// TIA Portal V18 program export: 17 tag tables, 4 data types, 7 data blocks, 10 code blocks (in call order from the OBs), 10 instance data blocks

VAR_GLOBAL   // PLC tag table "Cabinet_1"
   Sz1_Button_LED_ST25_ST26 AT %Q1100.0 : Bool;
   Sz1_Button_LED_ST26_ST27 AT %Q1100.1 : Bool;
   Sz1_Button_LED_ST24_ST23 AT %Q1100.2 : Bool;
   Sz1_Button_LED_ST23_ST22 AT %Q1100.3 : Bool;
   Sz1_Button_LED_Hyd_Up AT %Q1100.4 : Bool;
   Sz1_Button_LED_Hyd_Down AT %Q1100.5 : Bool;
   Sz1_Button_LED_Air_Up AT %Q1100.6 : Bool;
   Sz1_Button_LED_Air_Down AT %Q1100.7 : Bool;
   Sz1_Button_LED_Wibration AT %Q1101.0 : Bool;
   Sz1_Button_LED_SS_Down AT %Q1101.1 : Bool;
   Sz1_Button_LED_SS_Up AT %Q1101.2 : Bool;
   Sz1_Button_LED_SS_Drive_ST25 AT %Q1101.3 : Bool;
   Sz1_Button_LED_SS_Drive_ST24 AT %Q1101.4 : Bool;
   Sz1_Button_LED_SS_Drive_ST17 AT %Q1101.5 : Bool;
   Sz1_Button_LED_SS_Drive_ST14 AT %Q1101.6 : Bool;
   Reserved AT %Q1101.7 : Bool;
   Sz1_St25_SenA AT %I1100.0 : Bool;
   Sz1_St25_SenB AT %I1100.1 : Bool;
   Sz1_St25_SenC AT %I1100.2 : Bool;
   Sz1_St25_SenD AT %I1100.3 : Bool;
   Sz1_St26_SenA AT %I1100.4 : Bool;
   Sz1_St26_SenB AT %I1100.5 : Bool;
   Sz1_St26_SenC AT %I1100.6 : Bool;
   Sz1_St26_SenD AT %I1100.7 : Bool;
   Sz1_St23_SenA AT %I1101.0 : Bool;
   Sz1_St23_SenB AT %I1101.1 : Bool;
   Sz1_St23_SenC AT %I1101.2 : Bool;
   Sz1_St23_SenD AT %I1101.3 : Bool;
   Sz1_St24_SenA AT %I1101.4 : Bool;
   Sz1_St24_SenB AT %I1101.5 : Bool;
   Sz1_St24_SenC AT %I1101.6 : Bool;
   Sz1_St24_SenD AT %I1101.7 : Bool;
   Sz1_Button_ST25_ST26 AT %I1102.0 : Bool;
   Sz1_Button_ST26_ST27 AT %I1102.1 : Bool;
   Sz1_Button_ST24_ST23 AT %I1102.2 : Bool;
   Sz1_Button_ST23_ST22 AT %I1102.3 : Bool;
   Sz1_Button_Hyd_Up AT %I1102.4 : Bool;
   Sz1_Button_Hyd_Down AT %I1102.5 : Bool;
   Sz1_Button_Air_Up AT %I1102.6 : Bool;
   Sz1_Button_Air_Down AT %I1102.7 : Bool;
   Sz1_Button_Wibration AT %I1103.0 : Bool;
   Sz1_Button_SS_Down AT %I1103.1 : Bool;
   Sz1_Button_SS_Up AT %I1103.2 : Bool;
   Sz1_Button_SS_Drive_ST25 AT %I1103.3 : Bool;
   Sz1_Button_SS_Drive_ST24 AT %I1103.4 : Bool;
   Sz1_Button_SS_Drive_ST17 AT %I1103.5 : Bool;
   Sz1_Button_SS_Drive_ST14 AT %I1103.6 : Bool;
   "Reserved(1)" AT %I1103.7 : Bool;
   Sz1_Button_Wib_ST25 AT %I1104.0 : Bool;
   Sz1_Button_Wib_ST24 AT %I1104.1 : Bool;
   Sz1_Button_Wib_ST23 AT %I1104.2 : Bool;
   Sz1_Button_Centering_ST23 AT %I1104.3 : Bool;
   Sz1_Button_Centering_ST22 AT %I1104.4 : Bool;
   "Reserved(2)" AT %I1104.5 : Bool;
   "Reserved(3)" AT %I1104.6 : Bool;
   "Reserved(4)" AT %I1104.7 : Bool;
   Sz1_Button_LED_Centering_ST23 AT %Q1102.0 : Bool;
   Sz1_Button_LED_Centering_ST22 AT %Q1102.1 : Bool;
   "Reserved(5)" AT %Q1102.2 : Bool;
   "Reserved(6)" AT %Q1102.3 : Bool;
   "Reserved(7)" AT %Q1102.4 : Bool;
   "Reserved(8)" AT %Q1102.5 : Bool;
   "Reserved(9)" AT %Q1102.6 : Bool;
   "Reserved(10)" AT %Q1102.7 : Bool;
   Sz1_Safety1_1 AT %I1150.0 : Bool;
   "Reserved(11)" AT %I1150.1 : Bool;
   "Reserved(12)" AT %I1150.2 : Bool;
   "Reserved(13)" AT %I1150.3 : Bool;
   Sz1_Safety1_2 AT %I1150.4 : Bool;
   "Reserved(14)" AT %I1150.5 : Bool;
   "Reserved(15)" AT %I1150.6 : Bool;
   "Reserved(16)" AT %I1150.7 : Bool;
   "Reserved(17)" AT %I1151.0 : Bool;
   "Reserved(18)" AT %I1151.1 : Bool;
   "Reserved(19)" AT %I1151.2 : Bool;
   "Reserved(20)" AT %I1151.3 : Bool;
   "Reserved(21)" AT %I1151.4 : Bool;
   "Reserved(22)" AT %I1151.5 : Bool;
   "Reserved(23)" AT %I1151.6 : Bool;
   "Reserved(24)" AT %I1151.7 : Bool;
END_VAR

VAR_GLOBAL   // PLC tag table "Cabinet_10"
   Sz10_Button_LED_ST11_ST12 AT %Q2000.0 : Bool;
   Sz10_Button_LED_ST12_ST13 AT %Q2000.1 : Bool;
   "Reserved(146)" AT %Q2000.2 : Bool;
   "Reserved(147)" AT %Q2000.3 : Bool;
   "Reserved(148)" AT %Q2000.4 : Bool;
   "Reserved(149)" AT %Q2000.5 : Bool;
   "Reserved(150)" AT %Q2000.6 : Bool;
   "Reserved(151)" AT %Q2000.7 : Bool;
   Sz10_ST11_SenA AT %I2000.0 : Bool;
   Sz10_ST11_SenB AT %I2000.1 : Bool;
   Sz10_ST11_SenC AT %I2000.2 : Bool;
   Sz10_ST11_SenD AT %I2000.3 : Bool;
   Sz10_ST12_SenA AT %I2000.4 : Bool;
   Sz10_ST12_SenB AT %I2000.5 : Bool;
   Sz10_ST12_SenC AT %I2000.6 : Bool;
   Sz10_ST12_SenD AT %I2000.7 : Bool;
   Sz10_Button_ST11_ST12 AT %I2001.0 : Bool;
   Sz10_Button_ST12_ST13 AT %I2001.1 : Bool;
   "Reserved(152)" AT %I2001.2 : Bool;
   "Reserved(153)" AT %I2001.3 : Bool;
   "Reserved(154)" AT %I2001.4 : Bool;
   "Reserved(155)" AT %I2001.5 : Bool;
   "Reserved(156)" AT %I2001.6 : Bool;
   "Reserved(157)" AT %I2001.7 : Bool;
   Sz10_Safety1_1 AT %I2050.0 : Bool;
   "Reserved(158)" AT %I2050.1 : Bool;
   "Reserved(159)" AT %I2050.2 : Bool;
   "Reserved(160)" AT %I2050.3 : Bool;
   Sz10_Safety1_2 AT %I2050.4 : Bool;
   "Reserved(161)" AT %I2050.5 : Bool;
   "Reserved(162)" AT %I2050.6 : Bool;
   "Reserved(163)" AT %I2050.7 : Bool;
   "Reserved(171)" AT %I2051.0 : Bool;
   "Reserved(170)" AT %I2051.1 : Bool;
   "Reserved(169)" AT %I2051.2 : Bool;
   "Reserved(168)" AT %I2051.3 : Bool;
   "Reserved(167)" AT %I2051.4 : Bool;
   "Reserved(166)" AT %I2051.5 : Bool;
   "Reserved(165)" AT %I2051.6 : Bool;
   "Reserved(164)" AT %I2051.7 : Bool;
END_VAR

VAR_GLOBAL   // PLC tag table "Cabinet_11"
   Sz11_ST13_SenA AT %I2100.0 : Bool;
   Sz11_ST13_SenB AT %I2100.1 : Bool;
   Sz11_ST13_SenC AT %I2100.2 : Bool;
   Sz11_ST13_SenD AT %I2100.3 : Bool;
   Sz11_ST14_SenA AT %I2100.4 : Bool;
   Sz11_ST14_SenB AT %I2100.5 : Bool;
   Sz11_ST14_SenC AT %I2100.6 : Bool;
   Sz11_ST14_SenD AT %I2100.7 : Bool;
   Sz11_ST17_SenA AT %I2101.0 : Bool;
   Sz11_ST17_SenB AT %I2101.1 : Bool;
   Sz11_ST17_SenC AT %I2101.2 : Bool;
   Sz11_ST17_SenD AT %I2101.3 : Bool;
   "Reserved(188)" AT %I2101.4 : Bool;
   "Reserved(189)" AT %I2101.5 : Bool;
   "Reserved(190)" AT %I2101.6 : Bool;
   Sz11_Safety1_1 AT %I2150.0 : Bool;
   "Reserved(173)" AT %I2150.1 : Bool;
   "Reserved(174)" AT %I2150.2 : Bool;
   "Reserved(175)" AT %I2150.3 : Bool;
   Sz11_Safety1_2 AT %I2150.4 : Bool;
   "Reserved(176)" AT %I2150.5 : Bool;
   "Reserved(177)" AT %I2150.6 : Bool;
   "Reserved(178)" AT %I2150.7 : Bool;
   "Reserved(179)" AT %I2151.0 : Bool;
   "Reserved(180)" AT %I2151.1 : Bool;
   "Reserved(181)" AT %I2151.2 : Bool;
   "Reserved(182)" AT %I2151.3 : Bool;
   "Reserved(183)" AT %I2151.4 : Bool;
   "Reserved(184)" AT %I2151.5 : Bool;
   "Reserved(185)" AT %I2151.6 : Bool;
   "Reserved(186)" AT %I2151.7 : Bool;
   Sz11_Button_LED_ST13_ST14 AT %Q2100.0 : Bool;
   "Reserved(187)" AT %I2101.7 : Bool;
   Sz11_Button_LED_SS_Down AT %Q2100.1 : Bool;
   Sz11_Button_LED_SS_Up AT %Q2100.2 : Bool;
   Sz11_Button_LED_SS_Drive_ST14 AT %Q2100.3 : Bool;
   Sz11_Button_LED_SS_Drive_ST17 AT %Q2100.4 : Bool;
   Sz11_Button_LED_SS_Drive_ST24 AT %Q2100.5 : Bool;
   Sz11_Button_LED_SS_Drive_ST25 AT %Q2100.6 : Bool;
   "Reserved(172)" AT %Q2100.7 : Bool;
   Sz11_Button_ST13_ST14 AT %I2102.0 : Bool;
   Sz11_Button_SS_Down AT %I2102.1 : Bool;
   Sz11_Button_SS_Up AT %I2102.2 : Bool;
   Sz11_Button_SS_Drive_ST14 AT %I2102.3 : Bool;
   Sz11_Button_SS_Drive_ST17 AT %I2102.4 : Bool;
   Sz11_Button_SS_Drive_ST24 AT %I2102.5 : Bool;
   Sz11_Button_SS_Drive_ST25 AT %I2102.6 : Bool;
END_VAR

VAR_GLOBAL   // PLC tag table "Cabinet_2"
   Sz2_Button_LED_ST27_ST28 AT %Q1200.0 : Bool;
   Sz2_Button_LED_ST28_ST29 AT %Q1200.1 : Bool;
   Sz2_Button_LED_ST22_ST21 AT %Q1200.2 : Bool;
   Sz2_Button_LED_ST21_ST20 AT %Q1200.3 : Bool;
   Sz2_Button_LED_Centering_ST21 AT %Q1200.4 : Bool;
   Sz2_Button_LED_Centering_ST20 AT %Q1200.5 : Bool;
   "Reserved(25)" AT %Q1200.6 : Bool;
   "Reserved(26)" AT %Q1200.7 : Bool;
   Sz2_ST27_SenA AT %I1200.0 : Bool;
   Sz2_ST27_SenB AT %I1200.1 : Bool;
   Sz2_ST27_SenC AT %I1200.2 : Bool;
   Sz2_ST27_SenD AT %I1200.3 : Bool;
   Sz2_ST28_SenA AT %I1200.4 : Bool;
   Sz2_ST28_SenB AT %I1200.5 : Bool;
   Sz2_ST28_SenC AT %I1200.6 : Bool;
   Sz2_ST28_SenD AT %I1200.7 : Bool;
   Sz2_ST21_SenA AT %I1201.0 : Bool;
   Sz2_ST21_SenB AT %I1201.1 : Bool;
   Sz2_ST21_SenC AT %I1201.2 : Bool;
   Sz2_ST21_SenD AT %I1201.3 : Bool;
   Sz2_ST22_SenA AT %I1201.4 : Bool;
   Sz2_ST22_SenB AT %I1201.5 : Bool;
   Sz2_ST22_SenC AT %I1201.6 : Bool;
   Sz2_ST22_SenD AT %I1201.7 : Bool;
   Sz2_Button_ST27_ST28 AT %I1202.0 : Bool;
   Sz2_Button_ST28_ST29 AT %I1202.1 : Bool;
   Sz2_Button_ST22_ST21 AT %I1202.2 : Bool;
   Sz2_Button_ST21_ST20 AT %I1202.3 : Bool;
   Sz2_Button_Centering_ST21 AT %I1202.4 : Bool;
   Sz2_Button_Centering_ST20 AT %I1202.5 : Bool;
   "Reserved(27)" AT %I1202.6 : Bool;
   "Reserved(28)" AT %I1202.7 : Bool;
   Sz2_Safety_1_1 AT %I1250.0 : Bool;
   Sz2_Safety_1_2 AT %I1250.4 : Bool;
   "Reserved(29)" AT %I1250.1 : Bool;
   "Reserved(30)" AT %I1250.2 : Bool;
   "Reserved(31)" AT %I1250.3 : Bool;
   "Reserved(32)" AT %I1250.5 : Bool;
   "Reserved(33)" AT %I1250.6 : Bool;
   "Reserved(34)" AT %I1250.7 : Bool;
   "Reserved(35)" AT %I1251.0 : Bool;
   "Reserved(36)" AT %I1251.1 : Bool;
   "Reserved(37)" AT %I1251.2 : Bool;
   "Reserved(38)" AT %I1251.3 : Bool;
   "Reserved(39)" AT %I1251.4 : Bool;
   "Reserved(40)" AT %I1251.5 : Bool;
   "Reserved(41)" AT %I1251.6 : Bool;
   "Reserved(42)" AT %I1251.7 : Bool;
END_VAR

VAR_GLOBAL   // PLC tag table "Cabinet_3"
   Sz3_Button_LED_ST29_ST30 AT %Q1300.0 : Bool;
   Sz3_Button_LED_ST30_ST31 AT %Q1300.1 : Bool;
   Sz3_Button_LED_ST18_ST37 AT %Q1300.2 : Bool;
   Sz3_Button_LED_ST19_ST18 AT %Q1300.3 : Bool;
   Sz3_Button_LED_ST20_ST19 AT %Q1300.4 : Bool;
   Sz3_Button_LED_Centering_ST19 AT %Q1300.5 : Bool;
   Sz3_Button_LED_Centering_ST18 AT %Q1300.6 : Bool;
   "Reserved(43)" AT %Q1300.7 : Bool;
   Sz3_ST29_SenA AT %I1300.0 : Bool;
   Sz3_ST29_SenB AT %I1300.1 : Bool;
   Sz3_ST29_SenC AT %I1300.2 : Bool;
   Sz3_ST29_SenD AT %I1300.3 : Bool;
   Sz3_ST30_SenA AT %I1300.4 : Bool;
   Sz3_ST30_SenB AT %I1300.5 : Bool;
   Sz3_ST30_SenC AT %I1300.6 : Bool;
   Sz3_ST30_SenD AT %I1300.7 : Bool;
   Sz3_ST31_SenA AT %I1301.0 : Bool;
   Sz3_ST31_SenB AT %I1301.1 : Bool;
   Sz3_ST31_SenC AT %I1301.2 : Bool;
   Sz3_ST31_SenD AT %I1301.3 : Bool;
   Sz3_ST18_SenA AT %I1301.4 : Bool;
   Sz3_ST18_SenB AT %I1301.5 : Bool;
   Sz3_ST18_SenC AT %I1301.6 : Bool;
   Sz3_ST18_SenD AT %I1301.7 : Bool;
   Sz3_ST19_SenA AT %I1302.0 : Bool;
   Sz3_ST19_SenB AT %I1302.1 : Bool;
   Sz3_ST19_SenC AT %I1302.2 : Bool;
   Sz3_ST19_SenD AT %I1302.3 : Bool;
   Sz3_ST20_SenA AT %I1302.4 : Bool;
   Sz3_ST20_SenB AT %I1302.5 : Bool;
   Sz3_ST20_SenC AT %I1302.6 : Bool;
   Sz3_ST20_SenD AT %I1302.7 : Bool;
   Sz3_Button_ST29_ST30 AT %I1303.0 : Bool;
   Sz3_Button_ST30_ST31 AT %I1303.1 : Bool;
   Sz3_Button_ST31_ST32 AT %I1303.2 : Bool;
   Sz3_Button_ST18_ST37 AT %I1303.3 : Bool;
   Sz3_Button_ST19_ST18 AT %I1303.4 : Bool;
   Sz3_Button_ST20_ST19 AT %I1303.5 : Bool;
   Sz3_Button_Centering_ST19 AT %I1303.6 : Bool;
   Sz3_Button_Centering_ST18 AT %I1303.7 : Bool;
   Sz3_Safety1_1 AT %I1304.0 : Bool;
   "Reserved(44)" AT %I1304.1 : Bool;
   "Reserved(45)" AT %I1304.2 : Bool;
   "Reserved(46)" AT %I1304.3 : Bool;
   Sz3_Safety1_2 AT %I1304.4 : Bool;
   "Reserved(47)" AT %I1304.5 : Bool;
   "Reserved(48)" AT %I1304.6 : Bool;
   "Reserved(49)" AT %I1304.7 : Bool;
   "Reserved(50)" AT %I1305.0 : Bool;
   "Reserved(51)" AT %I1305.1 : Bool;
   "Reserved(52)" AT %I1305.2 : Bool;
   "Reserved(53)" AT %I1305.3 : Bool;
   "Reserved(54)" AT %I1305.4 : Bool;
   "Reserved(55)" AT %I1305.5 : Bool;
   "Reserved(56)" AT %I1305.6 : Bool;
   "Reserved(57)" AT %I1305.7 : Bool;
END_VAR

VAR_GLOBAL   // PLC tag table "Cabinet_4"
   Sz4_Button_LED_ST32_ST33 AT %Q1400.0 : Bool;
   Sz4_Button_LED_ST33_ST34 AT %Q1400.1 : Bool;
   Sz4_Button_LED_ST36_ST38 AT %Q1400.2 : Bool;
   Sz4_Button_LED_ST37_ST36 AT %Q1400.3 : Bool;
   Sz4_Button_LED_ST34_ST33 AT %Q1400.4 : Bool;
   Sz4_Button_LED_ST38_ST36 AT %Q1400.5 : Bool;
   "Reserved(58)" AT %Q1400.6 : Bool;
   "Reserved(59)" AT %Q1400.7 : Bool;
   Sz4_ST32_SenA AT %I1400.0 : Bool;
   Sz4_ST32_SenB AT %I1400.1 : Bool;
   Sz4_ST32_SenC AT %I1400.2 : Bool;
   Sz4_ST32_SenD AT %I1400.3 : Bool;
   Sz4_ST33_SenA AT %I1400.4 : Bool;
   Sz4_ST33_SenB AT %I1400.5 : Bool;
   Sz4_ST33_SenC AT %I1400.6 : Bool;
   Sz4_ST33_SenD AT %I1400.7 : Bool;
   Sz4_ST36_SenA AT %I1401.0 : Bool;
   Sz4_ST36_SenB AT %I1401.1 : Bool;
   Sz4_ST36_SenC AT %I1401.2 : Bool;
   Sz4_ST36_SenD AT %I1401.3 : Bool;
   Sz4_ST37_SenA AT %I1401.4 : Bool;
   Sz4_ST37_SenB AT %I1401.5 : Bool;
   Sz4_ST37_SenC AT %I1401.6 : Bool;
   Sz4_ST37_SenD AT %I1401.7 : Bool;
   Sz4_Button_ST32_ST33 AT %I1402.0 : Bool;
   Sz4_Button_ST33_ST34 AT %I1402.1 : Bool;
   Sz4_Button_ST36_ST38 AT %I1402.2 : Bool;
   Sz4_Button_ST37_ST36 AT %I1402.3 : Bool;
   Sz4_Button_ST34_ST33 AT %I1402.4 : Bool;
   Sz4_Button_ST38_ST36 AT %I1402.5 : Bool;
   "Reserved(60)" AT %I1402.6 : Bool;
   "Reserved(61)" AT %I1402.7 : Bool;
   Sz4_Safety1_1 AT %I1403.0 : Bool;
   "Reserved(62)" AT %I1403.1 : Bool;
   "Reserved(63)" AT %I1403.2 : Bool;
   "Reserved(64)" AT %I1403.3 : Bool;
   Sz4_Safety1_2 AT %I1403.4 : Bool;
   "Reserved(65)" AT %I1403.5 : Bool;
   "Reserved(66)" AT %I1403.6 : Bool;
   "Reserved(67)" AT %I1403.7 : Bool;
   "Reserved(75)" AT %I1404.0 : Bool;
   "Reserved(74)" AT %I1404.1 : Bool;
   "Reserved(73)" AT %I1404.2 : Bool;
   "Reserved(72)" AT %I1404.3 : Bool;
   "Reserved(71)" AT %I1404.4 : Bool;
   "Reserved(70)" AT %I1404.5 : Bool;
   "Reserved(69)" AT %I1404.6 : Bool;
   "Reserved(68)" AT %I1404.7 : Bool;
END_VAR

VAR_GLOBAL   // PLC tag table "Cabinet_5_6"
   Sz5_ST01_SenA AT %I1504.0 : Bool;
   Sz5_ST01_SenB AT %I1504.1 : Bool;
   Sz5_ST01_SenC AT %I1504.2 : Bool;
   Sz5_ST01_SenD AT %I1504.3 : Bool;
   Sz5_ST02_SenA AT %I1504.4 : Bool;
   Sz5_ST02_SenB AT %I1504.5 : Bool;
   Sz5_ST02_SenC AT %I1504.6 : Bool;
   Sz5_ST02_SenD AT %I1504.7 : Bool;
   Sz5_ST34_SenA AT %I1505.0 : Bool;
   Sz5_ST34_SenB AT %I1505.1 : Bool;
   Sz5_ST34_SenC AT %I1505.2 : Bool;
   Sz5_ST34_SenD AT %I1505.3 : Bool;
   Sz5_ST35_SenA AT %I1505.4 : Bool;
   Sz5_ST35_SenB AT %I1505.5 : Bool;
   Sz5_ST35_SenC AT %I1505.6 : Bool;
   Sz5_ST35_SenD AT %I1505.7 : Bool;
   Sz5_ST38_SenA AT %I1506.0 : Bool;
   Sz5_ST38_SenB AT %I1506.1 : Bool;
   Sz5_ST38_SenC AT %I1506.2 : Bool;
   Sz5_ST38_SenD AT %I1506.3 : Bool;
END_VAR

VAR_GLOBAL   // PLC tag table "Cabinet_7"
   Sz7_Button_LED_SS_Down AT %Q1700.0 : Bool;
   Sz7_Button_LED_SS_Up AT %Q1700.1 : Bool;
   Sz7_Button_LED_SS_Drive_ST35 AT %Q1700.2 : Bool;
   Sz7_Button_LED_SS_Drive_ST02 AT %Q1700.3 : Bool;
   Sz7_Button_LED_SS_Drive_ST03 AT %Q1700.4 : Bool;
   Sz7_Button_LED_SS_Drive_ST04 AT %Q1700.5 : Bool;
   Sz7_Button_LED_ST04_ST05 AT %Q1700.6 : Bool;
   Sz7_Button_LED_ST05_ST06 AT %Q1700.7 : Bool;
   "Reserved(76)" AT %Q1701.0 : Bool;
   "Reserved(77)" AT %Q1701.1 : Bool;
   "Reserved(78)" AT %Q1701.2 : Bool;
   "Reserved(79)" AT %Q1701.3 : Bool;
   "Reserved(80)" AT %Q1701.4 : Bool;
   "Reserved(81)" AT %Q1701.5 : Bool;
   "Reserved(82)" AT %Q1701.6 : Bool;
   "Reserved(83)" AT %Q1701.7 : Bool;
   Sz7_ST03_SenA AT %I1700.0 : Bool;
   Sz7_ST03_SenB AT %I1700.1 : Bool;
   Sz7_ST03_SenC AT %I1700.2 : Bool;
   Sz7_ST03_SenD AT %I1700.3 : Bool;
   Sz7_ST04_SenA AT %I1700.4 : Bool;
   Sz7_ST04_SenB AT %I1700.5 : Bool;
   Sz7_ST04_SenC AT %I1700.6 : Bool;
   Sz7_ST04_SenD AT %I1700.7 : Bool;
   Sz7_ST04_SenE AT %I1701.0 : Bool;
   Sz7_ST04_SenF AT %I1701.1 : Bool;
   Sz7_ST05_SenA AT %I1701.2 : Bool;
   Sz7_ST05_SenB AT %I1701.3 : Bool;
   Sz7_ST05_SenC AT %I1701.4 : Bool;
   Sz7_ST05_SenD AT %I1701.5 : Bool;
   "Reserved(84)" AT %I1701.6 : Bool;
   "Reserved(85)" AT %I1701.7 : Bool;
   Sz7_Button_SS_Down AT %I1702.0 : Bool;
   Sz7_Safety1_1 AT %I1750.0 : Bool;
   Sz7_Button_SS_Up AT %I1702.1 : Bool;
   Sz7_Button_SS_Drive_ST35 AT %I1702.2 : Bool;
   Sz7_Button_SS_Drive_ST02 AT %I1702.3 : Bool;
   Sz7_Button_SS_Drive_ST03 AT %I1702.4 : Bool;
   Sz7_Button_SS_Drive_ST04 AT %I1702.5 : Bool;
   Sz7_Button_ST04_ST05 AT %I1702.6 : Bool;
   Sz7_Button_ST05_ST06 AT %I1702.7 : Bool;
   "Reserved(100)" AT %I1703.0 : Bool;
   "Reserved(101)" AT %I1703.1 : Bool;
   "Reserved(102)" AT %I1703.2 : Bool;
   "Reserved(103)" AT %I1703.3 : Bool;
   "Reserved(104)" AT %I1703.4 : Bool;
   "Reserved(105)" AT %I1703.5 : Bool;
   "Reserved(106)" AT %I1703.6 : Bool;
   "Reserved(107)" AT %I1703.7 : Bool;
   "Reserved(86)" AT %I1750.1 : Bool;
   "Reserved(87)" AT %I1750.2 : Bool;
   "Reserved(88)" AT %I1750.3 : Bool;
   "Sz7-Safety1_2" AT %I1750.4 : Bool;
   "Reserved(89)" AT %I1750.5 : Bool;
   "Reserved(90)" AT %I1750.6 : Bool;
   "Reserved(91)" AT %I1750.7 : Bool;
   "Reserved(92)" AT %I1751.0 : Bool;
   "Reserved(93)" AT %I1751.1 : Bool;
   "Reserved(94)" AT %I1751.2 : Bool;
   "Reserved(95)" AT %I1751.3 : Bool;
   "Reserved(96)" AT %I1751.4 : Bool;
   "Reserved(97)" AT %I1751.5 : Bool;
   "Reserved(98)" AT %I1751.6 : Bool;
   "Reserved(99)" AT %I1751.7 : Bool;
END_VAR

VAR_GLOBAL   // PLC tag table "Cabinet_8"
   Sz8_Button_LED_ST06_ST07 AT %Q1800.0 : Bool;
   Sz8_Button_LED_ST07_ST08 AT %Q1800.1 : Bool;
   Sz8_Button_LED_ST08_ST09 AT %Q1800.2 : Bool;
   Sz8_Button_LED_Centering_ST08 AT %Q1800.3 : Bool;
   "Reserved(108)" AT %Q1800.4 : Bool;
   "Reserved(109)" AT %Q1800.5 : Bool;
   "Reserved(110)" AT %Q1800.6 : Bool;
   "Reserved(111)" AT %Q1800.7 : Bool;
   Sz8_ST06_SenA AT %I1800.0 : Bool;
   Sz8_ST06_SenB AT %I1800.1 : Bool;
   Sz8_ST06_SenC AT %I1800.2 : Bool;
   Sz8_ST06_SenD AT %I1800.3 : Bool;
   Sz8_ST07_SenA AT %I1800.4 : Bool;
   Sz8_ST07_SenB AT %I1800.5 : Bool;
   Sz8_ST07_SenC AT %I1800.6 : Bool;
   Sz8_ST07_SenD AT %I1800.7 : Bool;
   Sz8_ST08_SenA AT %I1801.0 : Bool;
   Sz8_ST08_SenB AT %I1801.1 : Bool;
   Sz8_ST08_SenC AT %I1801.2 : Bool;
   Sz8_ST08_SenD AT %I1801.3 : Bool;
   Sz8_Button_ST06_ST07 AT %I1801.4 : Bool;
   Sz8_Button_ST07_ST08 AT %I1801.5 : Bool;
   Sz8_Button_ST08_ST09 AT %I1801.6 : Bool;
   Sz8_Button_Centering_ST08 AT %I1801.7 : Bool;
   Sz8_Safety1_1 AT %I1850.0 : Bool;
   "Reserved(112)" AT %I1850.1 : Bool;
   "Reserved(113)" AT %I1850.2 : Bool;
   "Reserved(114)" AT %I1850.3 : Bool;
   Sz8_Safety1_2 AT %I1850.4 : Bool;
   "Reserved(115)" AT %I1850.5 : Bool;
   "Reserved(116)" AT %I1850.6 : Bool;
   "Reserved(117)" AT %I1850.7 : Bool;
   "Reserved(118)" AT %I1851.0 : Bool;
   "Reserved(119)" AT %I1851.1 : Bool;
   "Reserved(120)" AT %I1851.2 : Bool;
   "Reserved(121)" AT %I1851.3 : Bool;
   "Reserved(122)" AT %I1851.4 : Bool;
   "Reserved(123)" AT %I1851.5 : Bool;
   "Reserved(124)" AT %I1851.6 : Bool;
   "Reserved(125)" AT %I1851.7 : Bool;
END_VAR

VAR_GLOBAL   // PLC tag table "Cabinet_9"
   Sz9_Button_LED_ST09_ST10 AT %Q1900.0 : Bool;
   Sz9_Button_LED_ST10_ST11 AT %Q1900.1 : Bool;
   Sz9_ST09_SenA AT %I1900.0 : Bool;
   Sz9_ST09_SenB AT %I1900.1 : Bool;
   Sz9_ST09_SenC AT %I1900.2 : Bool;
   Sz9_ST09_SenD AT %I1900.3 : Bool;
   Sz9_ST10_SenA AT %I1900.4 : Bool;
   Sz9_ST10_SenB AT %I1900.5 : Bool;
   Sz9_ST10_SenC AT %I1900.6 : Bool;
   Sz9_ST10_SenD AT %I1900.7 : Bool;
   Sz9_Button_ST09_ST10 AT %I1901.0 : Bool;
   Sz9_Button_ST10_ST11 AT %I1901.1 : Bool;
   "Reserved(126)" AT %I1901.2 : Bool;
   "Reserved(127)" AT %I1901.3 : Bool;
   "Reserved(128)" AT %I1901.4 : Bool;
   "Reserved(129)" AT %I1901.5 : Bool;
   "Reserved(130)" AT %I1901.6 : Bool;
   "Reserved(131)" AT %I1901.7 : Bool;
   Sz9_Safety1_1 AT %I1950.0 : Bool;
   Sz9_Safety1_2 AT %I1950.4 : Bool;
   "Reserved(132)" AT %I1950.1 : Bool;
   "Reserved(133)" AT %I1950.2 : Bool;
   "Reserved(134)" AT %I1950.3 : Bool;
   "Reserved(135)" AT %I1950.5 : Bool;
   "Reserved(136)" AT %I1950.6 : Bool;
   "Reserved(137)" AT %I1950.7 : Bool;
   "Reserved(138)" AT %I1951.0 : Bool;
   "Reserved(139)" AT %I1951.1 : Bool;
   "Reserved(140)" AT %I1951.2 : Bool;
   "Reserved(141)" AT %I1951.3 : Bool;
   "Reserved(142)" AT %I1951.4 : Bool;
   "Reserved(143)" AT %I1951.5 : Bool;
   "Reserved(144)" AT %I1951.6 : Bool;
   "Reserved(145)" AT %I1951.7 : Bool;
END_VAR

VAR_GLOBAL   // PLC tag table "CentralShifter"
   iCS_SensorHoming_Left AT %I800.0 : Bool;
   iCS_SensorHoming_Right AT %I800.1 : Bool;
END_VAR

VAR_GLOBAL   // PLC tag table "Default tag table"
   CS_Drive_PL_Actor_Interface_AddressIn AT %I50.0 : "PD_TEL105_IN";
   CS_Drive_PL_Actor_Interface_AddressOut AT %Q50.0 : "PD_TEL105_OUT";
   CS_Drive_PP_Actor_Interface_AddressIn AT %I18.0 : "PD_TEL105_IN";
   CS_Drive_PP_Actor_Interface_AddressOut AT %Q18.0 : "PD_TEL105_OUT";
   CS_Drive_TL_Actor_Interface_AddressIn AT %I102.0 : "PD_TEL105_IN";
   CS_Drive_TL_Actor_Interface_AddressOut AT %Q102.0 : "PD_TEL105_OUT";
   CS_Drive_TP_Actor_Interface_AddressIn AT %I76.0 : "PD_TEL105_IN";
   CS_Drive_TP_Actor_Interface_AddressOut AT %Q76.0 : "PD_TEL105_OUT";
   ST23_PAL_Down AT %Q900.0 : Bool;
   ST23_PAL_Up AT %Q900.1 : Bool;
   ST23_MOD1_Up AT %Q900.2 : Bool;
   ST23_MOD2_Up AT %Q900.3 : Bool;
   ST23_MOD3_Up AT %Q900.4 : Bool;
   ST24_PAL_Down AT %Q900.5 : Bool;
   ST24_PAL_Up AT %Q900.6 : Bool;
   ST24_MOD1_Up AT %Q900.7 : Bool;
   ST24_MOD2_Up AT %Q901.0 : Bool;
   ST24_MOD3_Up AT %Q901.1 : Bool;
   ST25_PAL_Down AT %Q901.2 : Bool;
   ST25_PAL_Up AT %Q901.3 : Bool;
   ST25_MOD1_Up AT %Q901.4 : Bool;
   ST25_MOD2_Up AT %Q901.5 : Bool;
   ST25_MOD3_Up AT %Q901.6 : Bool;
   Reserve AT %Q901.7 : Bool;
   ST23_MOD1_Sen11 AT %I900.0 : Bool;
   ST23_MOD1_Sen12 AT %I900.1 : Bool;
   ST23_MOD1_Sen21 AT %I900.2 : Bool;
   ST23_MOD1_Sen22 AT %I900.3 : Bool;
   ST23_MOD2_Sen11 AT %I900.4 : Bool;
   ST23_MOD2_Sen12 AT %I900.5 : Bool;
   ST23_MOD2_Sen21 AT %I900.6 : Bool;
   ST23_MOD2_Sen22 AT %I900.7 : Bool;
   ST23_MOD3_Sen11 AT %I901.0 : Bool;
   ST23_MOD3_Sen12 AT %I901.1 : Bool;
   ST23_MOD3_Sen21 AT %I901.2 : Bool;
   ST23_MOD3_Sen22 AT %I901.3 : Bool;
   ST23_PAL_Sen11 AT %I901.4 : Bool;
   ST23_PAL_Sen12 AT %I901.5 : Bool;
   ST23_PAL_Sen21 AT %I901.6 : Bool;
   ST23_PAL_Sen22 AT %I901.7 : Bool;
   ST24_MOD1_Sen11 AT %I902.0 : Bool;
   ST24_MOD1_Sen12 AT %I902.1 : Bool;
   ST24_MOD1_Sen21 AT %I902.2 : Bool;
   ST24_MOD1_Sen22 AT %I902.3 : Bool;
   ST24_MOD2_Sen11 AT %I902.4 : Bool;
   ST24_MOD2_Sen12 AT %I902.5 : Bool;
   ST24_MOD2_Sen21 AT %I902.6 : Bool;
   ST24_MOD2_Sen22 AT %I902.7 : Bool;
   ST24_MOD3_Sen11 AT %I903.0 : Bool;
   ST24_MOD3_Sen12 AT %I903.1 : Bool;
   ST24_MOD3_Sen21 AT %I903.2 : Bool;
   ST24_MOD3_Sen22 AT %I903.3 : Bool;
   ST24_PAL_Sen11 AT %I903.4 : Bool;
   ST24_PAL_Sen12 AT %I903.5 : Bool;
   ST24_PAL_Sen21 AT %I903.6 : Bool;
   ST24_PAL_Sen22 AT %I903.7 : Bool;
   ST23_Rol_Up AT %Q902.0 : Bool;
   ST24_Rol_Up AT %Q902.1 : Bool;
   ST25_Rol_Up AT %Q902.2 : Bool;
   ST25_MOD1_Sen11 AT %I904.0 : Bool;
   ST25_MOD1_Sen12 AT %I904.1 : Bool;
   ST25_MOD1_Sen21 AT %I904.2 : Bool;
   ST25_MOD1_Sen22 AT %I904.3 : Bool;
   ST25_MOD2_Sen11 AT %I904.4 : Bool;
   ST25_MOD2_Sen12 AT %I904.5 : Bool;
   ST25_MOD2_Sen21 AT %I904.6 : Bool;
   ST25_MOD2_Sen22 AT %I904.7 : Bool;
   ST25_MOD3_Sen11 AT %I905.0 : Bool;
   ST25_MOD3_Sen12 AT %I905.1 : Bool;
   ST25_MOD3_Sen21 AT %I905.2 : Bool;
   ST25_MOD3_Sen22 AT %I905.3 : Bool;
   ST25_PAL_Sen11 AT %I905.4 : Bool;
   ST25_PAL_Sen12 AT %I905.5 : Bool;
   ST25_PAL_Sen21 AT %I905.6 : Bool;
   ST25_PAL_Sen22 AT %I905.7 : Bool;
   "90" AT %Q0.0 : Bool;
   Estop_SS2_ChA AT %I915.0 : Bool;
   Estop_SS2_ChB AT %I915.4 : Bool;
   ST23_25_Y0 AT %Q910.0 : Bool;
   ST23_25_M0 AT %Q910.1 : Bool;
END_VAR

VAR_GLOBAL   // PLC tag table "LSql_UserConstants"
END_VAR
VAR_GLOBAL CONSTANT   // user constants
   LSQL_NUMBER_OF_COLUMNS_MAX : UInt := 9;   // upper bound of array for expected columns (zero-based!)
   LSQL_NUMBER_OF_ROWS_MAX : UInt := 9;   // upper bound of array for expected rows (zero-based!)
   LSQL_NUMBER_OF_ROWS_PER_CYCLE : USInt := 0;   // number of rows to be deserialized per cycle (0 = all at once)
END_VAR

VAR_GLOBAL   // PLC tag table "S1_R1"
   S1_R1_Valve_Up AT %Q300.0 : Bool;
   S1_R1_Valve_Down AT %Q300.1 : Bool;
   S1_R1_Sen_Drv_1 AT %I300.0 : Bool;
   S1_R1_Sen_Drv_2 AT %I300.1 : Bool;
   S1_R1_Sen_Drv_3 AT %I300.2 : Bool;
   S1_R1_Sen_Drv_4 AT %I300.3 : Bool;
   S1_R1_Sen_Val1_Up AT %I300.4 : Bool;
   S1_R1_Sen_Val1_Down AT %I300.5 : Bool;
   S1_R1_Sen_Val2_Up AT %I300.6 : Bool;
   S1_R1_Sen_Val2_Down AT %I300.7 : Bool;
   S1_R1_Hyd_Filtr AT %I301.0 : Bool;
   S1_R1_Hyd_Empty AT %I301.1 : Bool;
   S1_R1_Safety1_1 AT %I350.0 : Bool;
   S1_R1_Safety2_1 AT %I350.1 : Bool;
   S1_R1_Safety3_1 AT %I350.2 : Bool;
   S1_R1_Safety4_1 AT %I350.3 : Bool;
   S1_R1_Safety1_2 AT %I351.0 : Bool;
   S1_R1_Safety2_2 AT %I351.1 : Bool;
   S1_R1_Safety3_2 AT %I351.2 : Bool;
   S1_R1_Safety4_2 AT %I351.3 : Bool;
END_VAR

VAR_GLOBAL   // PLC tag table "S1_R2"
   S1_R2_Valve_Up AT %Q400.0 : Bool;
   S1_R2_Valve_Down AT %Q400.1 : Bool;
   S1_R2_Sen_Drv_1 AT %Q400.2 : Bool;
   S1_R2_Sen_Drv_2 AT %Q400.3 : Bool;
   S1_R2_Sen_Drv_3 AT %Q400.4 : Bool;
   S1_R2_Sen_Drv_4 AT %Q400.5 : Bool;
   S1_R2_Sen_Val1_Up AT %Q400.6 : Bool;
   S1_R2_Sen_Val1_Down AT %Q400.7 : Bool;
   S1_R2_Sen_Val2_Up AT %Q401.0 : Bool;
   S1_R2_Sen_Val2_Down AT %Q401.1 : Bool;
   S1_R2_Hyd_Filtr AT %Q401.2 : Bool;
   S1_R2_Hyd_Empty AT %Q401.3 : Bool;
   S1_R2_Safety1_1 AT %I450.0 : Bool;
   S1_R2_Safety2_1 AT %I450.1 : Bool;
   S1_R2_Safety3_1 AT %I450.2 : Bool;
   S1_R2_Safety4_1 AT %I450.3 : Bool;
   S1_R2_Safety1_2 AT %I451.0 : Bool;
   S1_R2_Safety2_2 AT %I451.1 : Bool;
   S1_R2_Safety3_2 AT %I451.2 : Bool;
   S1_R2_Safety4_2 AT %I451.3 : Bool;
END_VAR

VAR_GLOBAL   // PLC tag table "S2_R1"
   S2_R1_Valve_Up AT %Q500.0 : Bool;
   S2_R1_Valve_Down AT %Q500.1 : Bool;
   S2_R1_Sen_Drv_1 AT %Q500.2 : Bool;
   S2_R1_Sen_Drv_2 AT %Q500.3 : Bool;
   S2_R1_Sen_Drv_3 AT %Q500.4 : Bool;
   S2_R1_Sen_Drv_4 AT %Q500.5 : Bool;
   S2_R1_Sen_Val1_Up AT %Q500.6 : Bool;
   S2_R1_Sen_Val1_Down AT %Q500.7 : Bool;
   S2_R1_Sen_Val2_Up AT %Q501.0 : Bool;
   S2_R1_Sen_Val2_Down AT %Q501.1 : Bool;
   S2_R1_Hyd_Filtr AT %Q501.2 : Bool;
   S2_R1_Hyd_Empty AT %Q501.3 : Bool;
   S2_R1_Safety1_1 AT %I550.0 : Bool;
   S2_R1_Safety2_1 AT %I550.1 : Bool;
   S2_R1_Safety3_1 AT %I550.2 : Bool;
   S2_R1_Safety4_1 AT %I550.3 : Bool;
   S2_R1_Safety1_2 AT %I550.4 : Bool;
   S2_R1_Safety2_2 AT %I550.5 : Bool;
   S2_R1_Safety3_2 AT %I550.6 : Bool;
   S2_R1_Safety4_2 AT %I550.7 : Bool;
END_VAR

VAR_GLOBAL   // PLC tag table "S2_R2"
   S2_R2_Valve_Up AT %Q600.0 : Bool;
   S2_R2_Valve_Down AT %Q600.1 : Bool;
   S2_R2_Sen_Drv_1 AT %Q600.2 : Bool;
   S2_R2_Sen_Drv_2 AT %Q600.3 : Bool;
   S2_R2_Sen_Drv_3 AT %Q600.4 : Bool;
   S2_R2_Sen_Drv_4 AT %Q600.5 : Bool;
   S2_R2_Sen_Val1_Up AT %Q600.6 : Bool;
   S2_R2_Sen_Val1_Down AT %Q600.7 : Bool;
   S2_R2_Sen_Val2_Up AT %Q601.0 : Bool;
   S2_R2_Sen_Val2_Down AT %Q601.1 : Bool;
   S2_R2_Hyd_Filtr AT %Q601.2 : Bool;
   S2_R2_Hyd_Empty AT %Q601.3 : Bool;
   S2_R2_Safety1_1 AT %I650.0 : Bool;
   S2_R2_Safety2_1 AT %I650.1 : Bool;
   S2_R2_Safety3_1 AT %I650.2 : Bool;
   S2_R2_Safety4_1 AT %I650.3 : Bool;
   S2_R2_Safety1_2 AT %I650.4 : Bool;
   S2_R2_Safety2_2 AT %I650.5 : Bool;
   S2_R2_Safety3_2 AT %I650.6 : Bool;
   S2_R2_Safety4_2 AT %I650.7 : Bool;
END_VAR

TYPE "Pallet"
   STRUCT
      IsSelected : Bool;
      Station_Current_Position : Array[1..2] of Int;
      Station_Next_Position : Array[1..2] of Int;
      Number_Of_Elements : Array[1..4] of Int;
   END_STRUCT;
END_TYPE

TYPE "Station"
   STRUCT
      SensorA : Bool;
      SensorB : Bool;
      SensorC : Bool;
      SensorD : Bool;
      IsEmpty : Bool;
      IsOccupied : Bool;
      Number : Bool;
   END_STRUCT;
END_TYPE

TYPE "typeSqlData"
TITLE = typeSqlData
// structure for SQL data received from SELECT command
   STRUCT
      tdsHeader { ExternalAccessible := 'False'; ExternalVisible := 'False'; ExternalWritable := 'False'} : "LSql_typePacketHeader";
      columnCount { ExternalAccessible := 'False'; ExternalVisible := 'False'; ExternalWritable := 'False'} : UInt;   // number of received columns
      columns { ExternalAccessible := 'False'; ExternalVisible := 'False'; ExternalWritable := 'False'} : Array[0.."LSQL_NUMBER_OF_COLUMNS_MAX"] of "LSql_typeColumn";
      rowDataStart { ExternalAccessible := 'False'; ExternalVisible := 'False'; ExternalWritable := 'False'} : UInt;   // start address byte of rowData in TDS telegram
      rowDataLength { ExternalAccessible := 'False'; ExternalVisible := 'False'; ExternalWritable := 'False'} : UDInt;   // area length of rowData in TDS telegram
      rowCount { ExternalAccessible := 'False'; ExternalVisible := 'False'; ExternalWritable := 'False'} : UDInt;   // number of rows
      rowOverflow { ExternalAccessible := 'False'; ExternalVisible := 'False'; ExternalWritable := 'False'} : Bool;   // true = more rows (RowCount) than available UDT tokenRows
      rows { ExternalAccessible := 'False'; ExternalVisible := 'False'; ExternalWritable := 'False'} : Array[0.."LSQL_NUMBER_OF_ROWS_MAX"] of "typeTokenRow";
      errorToken { ExternalAccessible := 'False'; ExternalVisible := 'False'; ExternalWritable := 'False'} : "LSql_typeErrorToken";
   END_STRUCT;
   // // tdsHeader."type" : type of TDS package (4 = Server Response)
   // // tdsHeader.status : status of the TDS package (1= last package, 0 = more packages follow)
   // // tdsHeader.length : length of the TDS response
   // // tdsHeader.spId : process id of the SQL server
   // // tdsHeader.packetID : id of one message for a paket
   // // tdsHeader.window : not used - should be ignored by user
END_TYPE

TYPE "typeTokenRow"
TITLE = typeTokenRow
// use case specific structure for TDS token row
   STRUCT
      Pressure { ExternalAccessible := 'False'; ExternalVisible := 'False'; ExternalWritable := 'False'} : Int;   // row value for column 'Amount'
      Temperature { ExternalAccessible := 'False'; ExternalVisible := 'False'; ExternalWritable := 'False'} : Int;   // row value for column 'Color'
   END_STRUCT;
END_TYPE

DATA_BLOCK "Global_DB"   // DB16
{ S7_Optimized_Access := 'TRUE' }
// stored: MemoryReserve 100
   VAR
      Auto : Bool;
      Manual : Bool;
      Maintenance : Bool;
   END_VAR
BEGIN
END_DATA_BLOCK

DATA_BLOCK "HMI_DB"   // DB15
{ S7_Optimized_Access := 'TRUE' }
// stored: MemoryReserve 100
   VAR
      CS_Homing : Bool;
      CS_PP_Reset : Bool;
      CS_PL_Reset : Bool;
      CS_TP_Reset : Bool;
      CS_TL_Reset : Bool;
      CS_Virtual_Reset : Bool;
      CS_Reset : Bool;
      CS_PP_Power : Bool;
      CS_PL_Power : Bool;
      CS_TP_Power : Bool;
      CS_TL_Power : Bool;
      CS_Virtual_Power : Bool;
      CS_Power : Bool;
   END_VAR
BEGIN
END_DATA_BLOCK

DATA_BLOCK "Pallets_Stations"   // DB11
{ S7_Optimized_Access := 'TRUE' }
// stored: MemoryReserve 100
   VAR
      Pallets : Array[1..24] of "Pallet";
      Stations : Array[1..4, 1..12] of "Station";
   END_VAR
BEGIN
END_DATA_BLOCK

DATA_BLOCK "SqlCommands"   // DB3
TITLE = SqlCommands
{ S7_Optimized_Access := 'TRUE' }
AUTHOR : SIEMENS SUP Applications
VERSION : 1.1
// DB for holding the command strings for a Tabular Data Stream command to a SQL database
// stored: MemoryReserve 0
   VAR
      currentSqlCommand { ExternalAccessible := 'False'; ExternalVisible := 'False'; ExternalWritable := 'False'} : USInt := 6;   // index of current SQL command to be executed (zero-based)
      sqlCommands { ExternalAccessible := 'False'; ExternalVisible := 'False'; ExternalWritable := 'False'} : Array[0..25] of String;   // array of SQL command strings
   END_VAR
BEGIN
   sqlCommands[0] := 'insert into PLCDATA_1 values (7,8, 9)';
   sqlCommands[1] := 'Update PLCDATA_1 set IntegerValue1 = 7, IntegerValue2 = 7, IntegerValue3 = 7 where IntegerValue2 = 7';
   sqlCommands[2] := 'Select IntegerValue1 from PLCDATA_1';
   sqlCommands[3] := 'Select Fruit from PLCDATA_2 where Amount != 0';
   sqlCommands[4] := 'Select Fruit from PLCDATA_2 where color = $'red$'';
   sqlCommands[5] := 'insert into PLCDATA_3 values (7, $'2020-01-01 10:23:24.125$')';
   sqlCommands[6] := 'SELECT TOP (3) * FROM PLCDATA ORDER BY Temperature';
   sqlCommands[7] := 'execute myProcedureIn @input1=30, @input2=6, @input3=84';
   sqlCommands[8] := 'execute myProcedureSelect';
   sqlCommands[9] := 'declare @myout1 char(30),  @myout2 int execute myProcedureInOut @in1=$'pear$', @in2=$'yellow$', @in3=3, @out1=@myout1 OUTPUT, @out2=@myout2 OUTPUT select @myout1 as $'myOut1$', @myOut2 as $'myOut2$'';
   sqlCommands[10] := 'INSERT INTO [dbo].[errors] ([Text]) VALUES ($'remotetest$')';
   sqlCommands[11] := 'SELECT TOP (10) ValueReal1, ValueReal2, ValueReal3, ValueReal4, ValueReal5, ValueReal6, ValueReal7, ValueReal8, ValueReal9 FROM TestJulian';
   sqlCommands[12] := 'SELECT * FROM KompressionLog ORDER BY StentNr';
   sqlCommands[13] := 'execute SelectProc1';
   sqlCommands[14] := 'insert into TestDateTime values ($'01.01.1990 12:00:00$')';
   sqlCommands[15] := 'exec SetDateTime @Input1 = $'07.30.1990 12:00:00$'';
   sqlCommands[16] := 'SELECT TOP (100) MesId, MesId2, MesId3 FROM TestJulian';
   sqlCommands[17] := 'SELECT TOP (1) DateTime FROM TestDateTime';
   sqlCommands[18] := 'SELECT TOP 2 * FROM FunctionTest ORDER BY ID';
   sqlCommands[19] := 'INSERT INTO [dbo].[FunctionTest] DEFAULT VALUES';
   sqlCommands[20] := 'use [SQLFromPLC] declare @myout1 bit  execute  NachtragDatensaetze @inDateiPfad= $'C:\Program Files\Microsoft SQL Server\MSSQL14.SQLEXPRESS\MSSQL\DATA\iO.csv$', @outDone=@myout1 OUTPUT select @myout1 as $'myOut1$'';
   sqlCommands[21] := 'UPDATE [dbo].[KompressionLog] SET LotNummer = $'Test234$' WHERE KammerId = $'3$'';
END_DATA_BLOCK

DATA_BLOCK "SqlConfig"   // DB7
TITLE = SqlConfig
{ S7_Optimized_Access := 'TRUE' }
AUTHOR : SIEMENS SUP Applications
VERSION : 1.1
// DB for providing the connection settings for a Tabuar Data Stream to a SQL database
// stored: MemoryReserve 100
   VAR
      connectionSettings { ExternalAccessible := 'False'; ExternalVisible := 'False'; ExternalWritable := 'False'} : "LSql_typeConnectionSettings";
      enableLSql { ExternalAccessible := 'False'; ExternalVisible := 'False'; ExternalWritable := 'False'} : Bool;   // enables LSql block (starts connection and login, waits for execute commands)
      diagnostics { ExternalWritable := 'False'} : "LSql_typeDiagnostics";
      executeSqlCommand { ExternalAccessible := 'False'; ExternalVisible := 'False'; ExternalWritable := 'False'} : Bool;   // trigger to execute a single sql command. EnableLSql must be true before triggering
   END_VAR
BEGIN
   connectionSettings.interfaceSettings.InterfaceId := 64;
   connectionSettings.interfaceSettings.ID := 16#10;
   connectionSettings.interfaceSettings.ActiveEstablished := true;
   connectionSettings.interfaceSettings.RemoteAddress.ADDR[1] := 10;
   connectionSettings.interfaceSettings.RemoteAddress.ADDR[2..3] := 30;
   connectionSettings.interfaceSettings.RemoteAddress.ADDR[4] := 222;
   connectionSettings.interfaceSettings.RemotePort := 1433;
   connectionSettings.loginInformation.userName := 'SQL_S71500';
   connectionSettings.loginInformation.password := 'SQL_S71500';
   connectionSettings.loginInformation.serverName := 'SQLEXPRESS';
   connectionSettings.loginInformation.databaseName := 'S71500SQLDB';
END_DATA_BLOCK

DATA_BLOCK "SqlData"   // DB5
TITLE = SqlData
{ S7_Optimized_Access := 'TRUE' }
AUTHOR : SIEMENS SUP Applications
VERSION : 3.0
// DB for holding the strucutured data received from a Tabular Data Stream SELECT response
// stored: MemoryReserve 0
   VAR
      data { ExternalAccessible := 'False'; ExternalVisible := 'False'; ExternalWritable := 'False'} : "typeSqlData";
   END_VAR
BEGIN
END_DATA_BLOCK

DATA_BLOCK "SqlTdsReceive"   // DB8
TITLE = SqlTdsReceive
{ S7_Optimized_Access := 'TRUE'; DB_Accessible_From_OPC_UA := 'FALSE' }
AUTHOR : SIEMENS SUP Applications
VERSION : 3.0
// DB for holding the received data array of byte from a Tabular Data Stream (TDS) command to a SQL database
// stored: DBAccessibleFromOPCUA false, MemoryReserve 0
   VAR
      tdsTelegramArrayLength { ExternalAccessible := 'False'; ExternalVisible := 'False'; ExternalWritable := 'False'} : UDInt;   // number of Bytes received by TDS telegram and TRCV input
      tdsTelegramArray { ExternalAccessible := 'False'; ExternalVisible := 'False'; ExternalWritable := 'False'} : Array[0..9999] of Byte;   // array of Bytes of reconstructed TDS telegram
   END_VAR
BEGIN
END_DATA_BLOCK

ORGANIZATION_BLOCK "Main"   // OB1, LAD, ProgramCycle
TITLE = "Main Program Sweep (Cycle)"
{ S7_Optimized_Access := 'TRUE' }
// stored: SetENOAutomatically false
   VAR_INPUT
      Initial_Call : Bool;   // Initial call of this OB
      Remanence : Bool;   // =True, if remanent data are available
   END_VAR
BEGIN

REGION Network 1
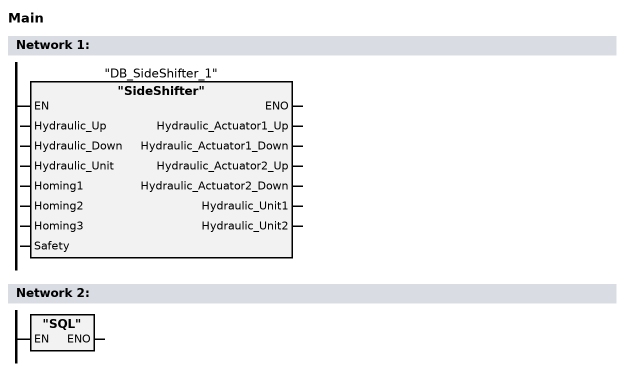
   RUNG wire#powerrail
      "DB_SideShifter_1"(Hydraulic_Up :=, Hydraulic_Down :=, Hydraulic_Unit :=, Homing1 :=, Homing2 :=, Homing3 :=, Safety :=, Hydraulic_Actuator1_Up =>, Hydraulic_Actuator1_Down =>, Hydraulic_Actuator2_Up =>, Hydraulic_Actuator2_Down =>, Hydraulic_Unit1 =>, Hydraulic_Unit2 =>)
   END_RUNG
   // the same network as SCL:
   "DB_SideShifter_1"();   // "SideShifter"
END_REGION

REGION Network 2
   RUNG wire#powerrail
      "SQL"()
   END_RUNG
   // the same network as SCL:
   "SQL"();
END_REGION
END_ORGANIZATION_BLOCK

FUNCTION_BLOCK "SideShifter"   // FB2, LAD
{ S7_Optimized_Access := 'TRUE' }
// stored: MemoryReserve 100, SetENOAutomatically false
   VAR_INPUT
      Hydraulic_Up : Bool;
      Hydraulic_Down : Bool;
      Hydraulic_Unit : Bool;
      Homing1 : Bool;
      Homing2 : Bool;
      Homing3 : Bool;
      Safety : Bool;
   END_VAR
   VAR_OUTPUT
      Hydraulic_Actuator1_Up : Bool;
      Hydraulic_Actuator1_Down : Bool;
      Hydraulic_Actuator2_Up : Bool;
      Hydraulic_Actuator2_Down : Bool;
      Hydraulic_Unit1 : Bool;
      Hydraulic_Unit2 : Bool;
   END_VAR
BEGIN
END_FUNCTION_BLOCK

FUNCTION "SQL" : Void   // FC2, LAD
{ S7_Optimized_Access := 'TRUE' }
// stored: SetENOAutomatically false
   VAR_TEMP
      tempDataReceived : Bool;   // temp flag for 'dataReceived' from FB 'LSql_Microsoft'
      tempAnalyzeDone : Bool;   // temp flag for 'done' from FB 'AnalyzeTokens'
      tempMetaDataAndRowsAvailable : Bool;   // temp flag for 'metaDataAndRowsAvailable' from FB 'AnalyzeTokens'
   END_VAR
BEGIN

REGION Network 1: TDS Connection and Communication Handling
   // this network handles the TDS connection and communication
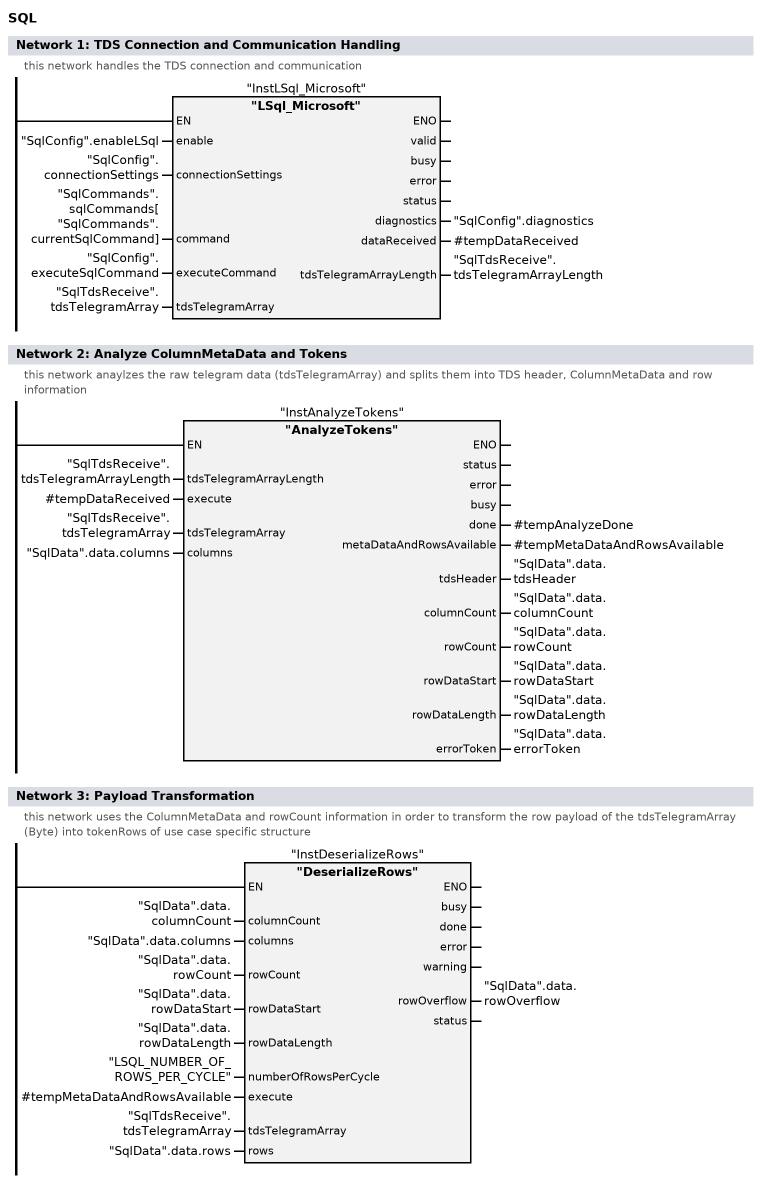
   RUNG wire#powerrail
      "InstLSql_Microsoft"(enable := "SqlConfig".enableLSql, connectionSettings := "SqlConfig".connectionSettings, command := "SqlCommands".sqlCommands["SqlCommands".currentSqlCommand], executeCommand := "SqlConfig".executeSqlCommand, tdsTelegramArray := "SqlTdsReceive".tdsTelegramArray, valid =>, busy =>, error =>, status =>, diagnostics => "SqlConfig".diagnostics, dataReceived => #tempDataReceived, tdsTelegramArrayLength => "SqlTdsReceive".tdsTelegramArrayLength)
   END_RUNG
   // the same network as SCL:
   "InstLSql_Microsoft"(enable := "SqlConfig".enableLSql,   // "LSql_Microsoft"
                        connectionSettings := "SqlConfig".connectionSettings,
                        command := "SqlCommands".sqlCommands["SqlCommands".currentSqlCommand],
                        executeCommand := "SqlConfig".executeSqlCommand,
                        tdsTelegramArray := "SqlTdsReceive".tdsTelegramArray,
                        diagnostics => "SqlConfig".diagnostics,
                        dataReceived => #tempDataReceived,
                        tdsTelegramArrayLength => "SqlTdsReceive".tdsTelegramArrayLength);
END_REGION

REGION Network 2: Analyze ColumnMetaData and Tokens
   // this network anaylzes the raw telegram data (tdsTelegramArray) and splits them into TDS header, ColumnMetaData and row information
   RUNG wire#powerrail
      "InstAnalyzeTokens"(tdsTelegramArrayLength := "SqlTdsReceive".tdsTelegramArrayLength, execute := #tempDataReceived, tdsTelegramArray := "SqlTdsReceive".tdsTelegramArray, columns := "SqlData".data.columns, status =>, error =>, busy =>, done => #tempAnalyzeDone, metaDataAndRowsAvailable => #tempMetaDataAndRowsAvailable, tdsHeader => "SqlData".data.tdsHeader, columnCount => "SqlData".data.columnCount, rowCount => "SqlData".data.rowCount, rowDataStart => "SqlData".data.rowDataStart, rowDataLength => "SqlData".data.rowDataLength, errorToken => "SqlData".data.errorToken)
   END_RUNG
   // the same network as SCL:
   "InstAnalyzeTokens"(tdsTelegramArrayLength := "SqlTdsReceive".tdsTelegramArrayLength,   // "AnalyzeTokens"
                       execute := #tempDataReceived,
                       tdsTelegramArray := "SqlTdsReceive".tdsTelegramArray,
                       columns := "SqlData".data.columns,
                       done => #tempAnalyzeDone,
                       metaDataAndRowsAvailable => #tempMetaDataAndRowsAvailable,
                       tdsHeader => "SqlData".data.tdsHeader,
                       columnCount => "SqlData".data.columnCount,
                       rowCount => "SqlData".data.rowCount,
                       rowDataStart => "SqlData".data.rowDataStart,
                       rowDataLength => "SqlData".data.rowDataLength,
                       errorToken => "SqlData".data.errorToken);
END_REGION

REGION Network 3: Payload Transformation
   // this network uses the ColumnMetaData and rowCount information in order to transform the row payload of the tdsTelegramArray (Byte) into tokenRows of use case specific structure
   RUNG wire#powerrail
      "InstDeserializeRows"(columnCount := "SqlData".data.columnCount, columns := "SqlData".data.columns, rowCount := "SqlData".data.rowCount, rowDataStart := "SqlData".data.rowDataStart, rowDataLength := "SqlData".data.rowDataLength, numberOfRowsPerCycle := "LSQL_NUMBER_OF_ROWS_PER_CYCLE", execute := #tempMetaDataAndRowsAvailable, tdsTelegramArray := "SqlTdsReceive".tdsTelegramArray, rows := "SqlData".data.rows, busy =>, done =>, error =>, warning =>, rowOverflow => "SqlData".data.rowOverflow, status =>)
   END_RUNG
   // the same network as SCL:
   "InstDeserializeRows"(columnCount := "SqlData".data.columnCount,   // "DeserializeRows"
                         columns := "SqlData".data.columns,
                         rowCount := "SqlData".data.rowCount,
                         rowDataStart := "SqlData".data.rowDataStart,
                         rowDataLength := "SqlData".data.rowDataLength,
                         numberOfRowsPerCycle := "LSQL_NUMBER_OF_ROWS_PER_CYCLE",
                         execute := #tempMetaDataAndRowsAvailable,
                         tdsTelegramArray := "SqlTdsReceive".tdsTelegramArray,
                         rows := "SqlData".data.rows,
                         rowOverflow => "SqlData".data.rowOverflow);
END_REGION
END_FUNCTION

FUNCTION_BLOCK "Pallet_Status"   // FB8, LAD
{ S7_Optimized_Access := 'TRUE' }
// stored: MemoryReserve 100, SetENOAutomatically false
   VAR_INPUT
      SensorA : Bool;
      SensorB : Bool;
      SensorC : Bool;
      SensorD : Bool;
   END_VAR
BEGIN
END_FUNCTION_BLOCK

FUNCTION_BLOCK "Pallets_Transport_System"   // FB9, LAD
{ S7_Optimized_Access := 'TRUE' }
// stored: MemoryReserve 100, SetENOAutomatically false
   VAR
      NumberOfPallet { S7_SetPoint := 'True'} : Int;
      Map : Array[1..4, 1..12] of Bool;
      MoveDirection : Int;   // 1-L, 2-Up, 3-R, 4-Down
      FoundSelectedPallet : Bool;
      CanMove : Bool;
   END_VAR
   VAR_TEMP
      i : Int;
      j : Int;
      k : Int;
   END_VAR
BEGIN

REGION Network 1 (SCL)
   // Sprawdzenie, które elementy sa wybrane i nadanie im nowej pozycji
   FOR #k := 1 TO 24 DO
       IF "Pallets_Stations".Pallets[#k].IsSelected THEN
           EXIT;
       END_IF;

   END_FOR;

   FOR #i := 1 TO 4 DO
       FOR #j := 1 TO 12 DO
           IF "Pallets_Stations".Pallets[#k].IsSelected THEN

               "Pallets_Stations".Pallets[#k].Station_Next_Position := "Pallets_Stations".Pallets[#k].Station_Current_Position;  // Initialisation

               CASE #MoveDirection OF
                   1:
                       IF "Pallets_Stations".Pallets[#k].Station_Next_Position[2] > 1 THEN  // Check Left
                           "Pallets_Stations".Pallets[#k].Station_Next_Position[2] := "Pallets_Stations".Pallets[#k].Station_Next_Position[2] - 1;
                       ELSE
                           #CanMove := FALSE;
                       END_IF;
                   3:
                       IF ("Pallets_Stations".Pallets[#k].Station_Next_Position[2] < 12) AND // Check Right
                           (("Pallets_Stations".Pallets[#k].Station_Next_Position[1] = 2 AND "Pallets_Stations".Pallets[#k].Station_Next_Position[2] < 12) OR ("Pallets_Stations".Pallets[#k].Station_Next_Position[1] <> 2 AND "Pallets_Stations".Pallets[#k].Station_Next_Position[2] < 11)) THEN
                           "Pallets_Stations".Pallets[#k].Station_Next_Position[2] := "Pallets_Stations".Pallets[#k].Station_Next_Position[2] + 1;
                       ELSE
                           #CanMove := FALSE;
                       END_IF;
                   2:
                       IF ("Pallets_Stations".Pallets[#k].Station_Next_Position[2] = 1) OR
                           (("Pallets_Stations".Pallets[#k].Station_Next_Position[1] = 1 AND "Pallets_Stations".Pallets[#k].Station_Next_Position[2] = 11) OR
                           ("Pallets_Stations".Pallets[#k].Station_Next_Position[1] = 2 AND "Pallets_Stations".Pallets[#k].Station_Next_Position[2] = 12) OR
                           ("Pallets_Stations".Pallets[#k].Station_Next_Position[1] = 3 AND "Pallets_Stations".Pallets[#k].Station_Next_Position[2] = 11) OR
                           ("Pallets_Stations".Pallets[#k].Station_Next_Position[1] = 4 AND "Pallets_Stations".Pallets[#k].Station_Next_Position[2] = 11)) THEN
                           IF "Pallets_Stations".Pallets[#k].Station_Next_Position[1] > 1 THEN
                               // Ruch w ostatniej kolumnie
                               IF "Pallets_Stations".Pallets[#k].Station_Next_Position[1] = 2 AND "Pallets_Stations".Pallets[#k].Station_Next_Position[2] = 12 THEN
                                   "Pallets_Stations".Pallets[#k].Station_Next_Position[1] := 1;
                                   "Pallets_Stations".Pallets[#k].Station_Next_Position[2] := 11;
                               ELSE
                                   "Pallets_Stations".Pallets[#k].Station_Next_Position[1] := "Pallets_Stations".Pallets[#k].Station_Next_Position[1] - 1;
                               END_IF;
                           ELSE
                               #CanMove := FALSE;
                           END_IF;
                       ELSE
                           #CanMove := FALSE;
                       END_IF;
                   4:
                       IF ("Pallets_Stations".Pallets[#k].Station_Next_Position[2] = 1) OR
                           (("Pallets_Stations".Pallets[#k].Station_Next_Position[1] = 1 AND "Pallets_Stations".Pallets[#k].Station_Next_Position[2] = 11) OR
                           ("Pallets_Stations".Pallets[#k].Station_Next_Position[1] = 2 AND "Pallets_Stations".Pallets[#k].Station_Next_Position[2] = 12) OR
                           ("Pallets_Stations".Pallets[#k].Station_Next_Position[1] = 3 AND "Pallets_Stations".Pallets[#k].Station_Next_Position[2] = 11) OR
                           ("Pallets_Stations".Pallets[#k].Station_Next_Position[1] = 4 AND "Pallets_Stations".Pallets[#k].Station_Next_Position[2] = 11)) THEN
                           IF "Pallets_Stations".Pallets[#k].Station_Next_Position[1] < 4 THEN
                               // Ruch w ostatniej kolumnie
                               IF "Pallets_Stations".Pallets[#k].Station_Next_Position[1] = 1 AND "Pallets_Stations".Pallets[#k].Station_Next_Position[2] = 11 THEN
                                   "Pallets_Stations".Pallets[#k].Station_Next_Position[1] := 2;
                                   "Pallets_Stations".Pallets[#k].Station_Next_Position[2] := 12;
                               ELSE
                                   "Pallets_Stations".Pallets[#k].Station_Next_Position[1] := "Pallets_Stations".Pallets[#k].Station_Next_Position[1] + 1;
                               END_IF;
                           ELSE
                               #CanMove := FALSE;
                           END_IF;
                       ELSE
                           #CanMove := FALSE;
                       END_IF;
               END_CASE;


               //TO DO Movement


               IF "Pallets_Stations".Stations["Pallets_Stations".Pallets[#k].Station_Next_Position[1], "Pallets_Stations".Pallets[#k].Station_Next_Position[2]].IsEmpty THEN
                   // Aktualizacja stanu stanowisk i palet


                   // Aktualizacja pozycji palety
                   "Pallets_Stations".Pallets[#k].Station_Current_Position := "Pallets_Stations".Pallets[#k].Station_Next_Position;
                   #CanMove := TRUE;
               ELSE
                   #CanMove := FALSE;  // Nowe stanowisko zajęte
               END_IF;


           END_IF;
       END_FOR;
   END_FOR;
END_REGION
END_FUNCTION_BLOCK

FUNCTION_BLOCK "CentralShifter"   // FB10, LAD
{ S7_Optimized_Access := 'TRUE' }
// stored: MemoryReserve 100, SetENOAutomatically false
   VAR
      MC_POWER_CS_PP { S7_SetPoint := 'True'} : MC_POWER;
      MC_POWER_CS_PL { S7_SetPoint := 'True'} : MC_POWER;
      MC_POWER_CS_TP { S7_SetPoint := 'True'} : MC_POWER;
      MC_POWER_CS_TL { S7_SetPoint := 'True'} : MC_POWER;
      MC_POWER_CS_Virtual { S7_SetPoint := 'True'} : MC_POWER;
      MC_RESET_CS_PP { S7_SetPoint := 'True'} : MC_RESET;
      MC_RESET_CS_PL { S7_SetPoint := 'True'} : MC_RESET;
      MC_RESET_CS_TP { S7_SetPoint := 'True'} : MC_RESET;
      MC_RESET_CS_TL { S7_SetPoint := 'True'} : MC_RESET;
      MC_GEARIN_CS_PP { S7_SetPoint := 'True'} : MC_GEARIN;
      MC_GEARIN_CS_PL { S7_SetPoint := 'True'} : MC_GEARIN;
      MC_GEARIN_CS_TP { S7_SetPoint := 'True'} : MC_GEARIN;
      MC_GEARIN_CS_TL { S7_SetPoint := 'True'} : MC_GEARIN;
      MC_HOME_CS_PP { S7_SetPoint := 'True'} : MC_HOME;
      MC_HOME_CS_PL { S7_SetPoint := 'True'} : MC_HOME;
      MC_HOME_CS_TP { S7_SetPoint := 'True'} : MC_HOME;
      MC_HOME_CS_TL { S7_SetPoint := 'True'} : MC_HOME;
      MC_RESET_CS_Virtual { S7_SetPoint := 'True'} : MC_RESET;
      MC_MOVEJOG_CS_PL { S7_SetPoint := 'True'} : MC_MOVEJOG;
      MC_HOME_CS_Virtual { S7_SetPoint := 'True'} : MC_HOME;
      MC_MOVEJOG_CS_PP { S7_SetPoint := 'True'} : MC_MOVEJOG;
      MC_MOVEJOG_CS_TL { S7_SetPoint := 'True'} : MC_MOVEJOG;
      MC_MOVEJOG_CS_TP { S7_SetPoint := 'True'} : MC_MOVEJOG;
      MC_MOVEJOG_CS_Virtual { S7_SetPoint := 'True'} : MC_MOVEJOG;
      MC_MOVERELATIVE_CS_Virtual { S7_SetPoint := 'True'} : MC_MOVERELATIVE;
      MC_MOVEABSOLUTE_CS_Virtual { S7_SetPoint := 'True'} : MC_MOVEABSOLUTE;
      Homeing_Status { S7_SetPoint := 'True'} : Int;
      Jog_Backward_Home : Bool;
      Jog_Forward_Home : Bool;
      Jog_Velocity : Int;
   END_VAR
BEGIN

REGION Network 1
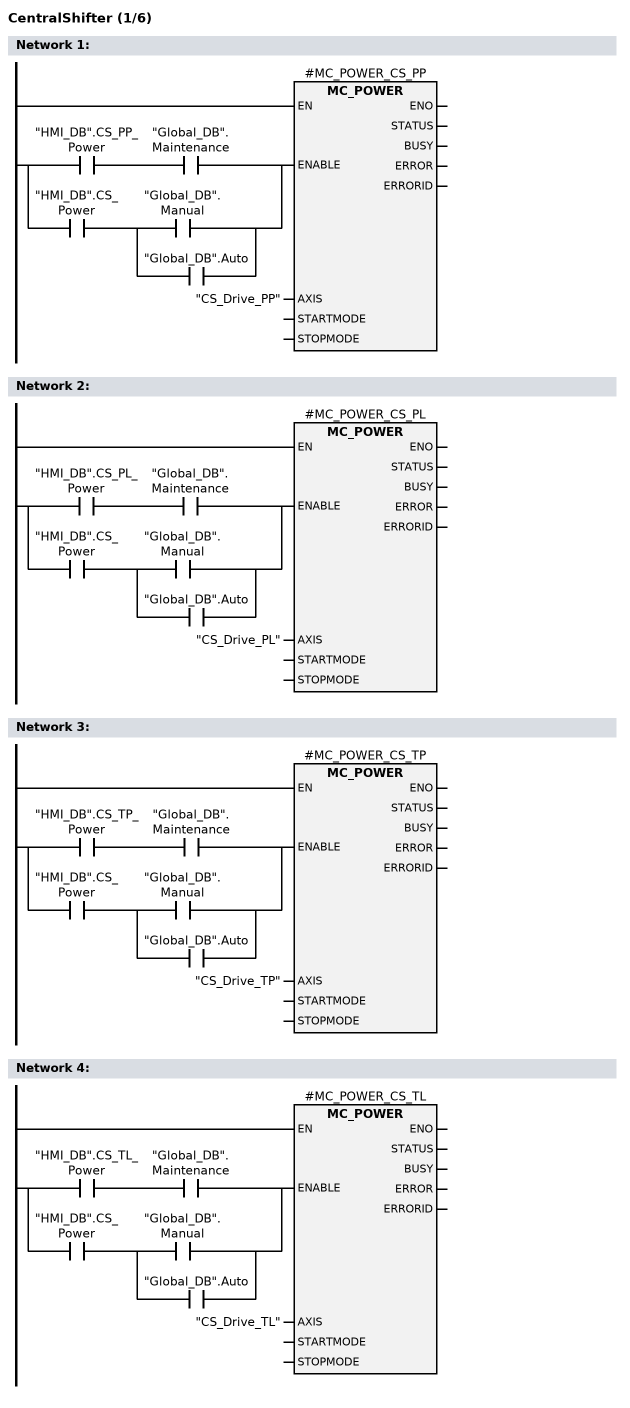
   RUNG wire#powerrail
      #MC_POWER_CS_PP.MC_POWER(Enable := wire#w2, Axis := "CS_Drive_PP", StartMode :=, StopMode :=, Status =>, Busy =>, Error =>, ErrorId =>)
   END_RUNG
   RUNG wire#powerrail
      Contact( "HMI_DB".CS_PP_Power )
      Contact( "Global_DB".Maintenance )
   END_RUNG wire#w2
   RUNG wire#powerrail
      Contact( "HMI_DB".CS_Power )
      wire#w1
      Contact( "Global_DB".Manual )
   END_RUNG wire#w2
   RUNG wire#w1
      Contact( "Global_DB".Auto )
   END_RUNG wire#w2
   // the same network as SCL:
   #MC_POWER_CS_PP(Enable := ("HMI_DB".CS_PP_Power AND "Global_DB".Maintenance) OR ("HMI_DB".CS_Power AND ("Global_DB".Manual OR "Global_DB".Auto)),   // MC_POWER
                   Axis := "CS_Drive_PP");
END_REGION

REGION Network 2
   RUNG wire#powerrail
      #MC_POWER_CS_PL.MC_POWER(Enable := wire#w2, Axis := "CS_Drive_PL", StartMode :=, StopMode :=, Status =>, Busy =>, Error =>, ErrorId =>)
   END_RUNG
   RUNG wire#powerrail
      Contact( "HMI_DB".CS_PL_Power )
      Contact( "Global_DB".Maintenance )
   END_RUNG wire#w2
   RUNG wire#powerrail
      Contact( "HMI_DB".CS_Power )
      wire#w1
      Contact( "Global_DB".Manual )
   END_RUNG wire#w2
   RUNG wire#w1
      Contact( "Global_DB".Auto )
   END_RUNG wire#w2
   // the same network as SCL:
   #MC_POWER_CS_PL(Enable := ("HMI_DB".CS_PL_Power AND "Global_DB".Maintenance) OR ("HMI_DB".CS_Power AND ("Global_DB".Manual OR "Global_DB".Auto)),   // MC_POWER
                   Axis := "CS_Drive_PL");
END_REGION

REGION Network 3
   RUNG wire#powerrail
      #MC_POWER_CS_TP.MC_POWER(Enable := wire#w2, Axis := "CS_Drive_TP", StartMode :=, StopMode :=, Status =>, Busy =>, Error =>, ErrorId =>)
   END_RUNG
   RUNG wire#powerrail
      Contact( "HMI_DB".CS_TP_Power )
      Contact( "Global_DB".Maintenance )
   END_RUNG wire#w2
   RUNG wire#powerrail
      Contact( "HMI_DB".CS_Power )
      wire#w1
      Contact( "Global_DB".Manual )
   END_RUNG wire#w2
   RUNG wire#w1
      Contact( "Global_DB".Auto )
   END_RUNG wire#w2
   // the same network as SCL:
   #MC_POWER_CS_TP(Enable := ("HMI_DB".CS_TP_Power AND "Global_DB".Maintenance) OR ("HMI_DB".CS_Power AND ("Global_DB".Manual OR "Global_DB".Auto)),   // MC_POWER
                   Axis := "CS_Drive_TP");
END_REGION

REGION Network 4
   RUNG wire#powerrail
      #MC_POWER_CS_TL.MC_POWER(Enable := wire#w2, Axis := "CS_Drive_TL", StartMode :=, StopMode :=, Status =>, Busy =>, Error =>, ErrorId =>)
   END_RUNG
   RUNG wire#powerrail
      Contact( "HMI_DB".CS_TL_Power )
      Contact( "Global_DB".Maintenance )
   END_RUNG wire#w2
   RUNG wire#powerrail
      Contact( "HMI_DB".CS_Power )
      wire#w1
      Contact( "Global_DB".Manual )
   END_RUNG wire#w2
   RUNG wire#w1
      Contact( "Global_DB".Auto )
   END_RUNG wire#w2
   // the same network as SCL:
   #MC_POWER_CS_TL(Enable := ("HMI_DB".CS_TL_Power AND "Global_DB".Maintenance) OR ("HMI_DB".CS_Power AND ("Global_DB".Manual OR "Global_DB".Auto)),   // MC_POWER
                   Axis := "CS_Drive_TL");
END_REGION

REGION Network 5
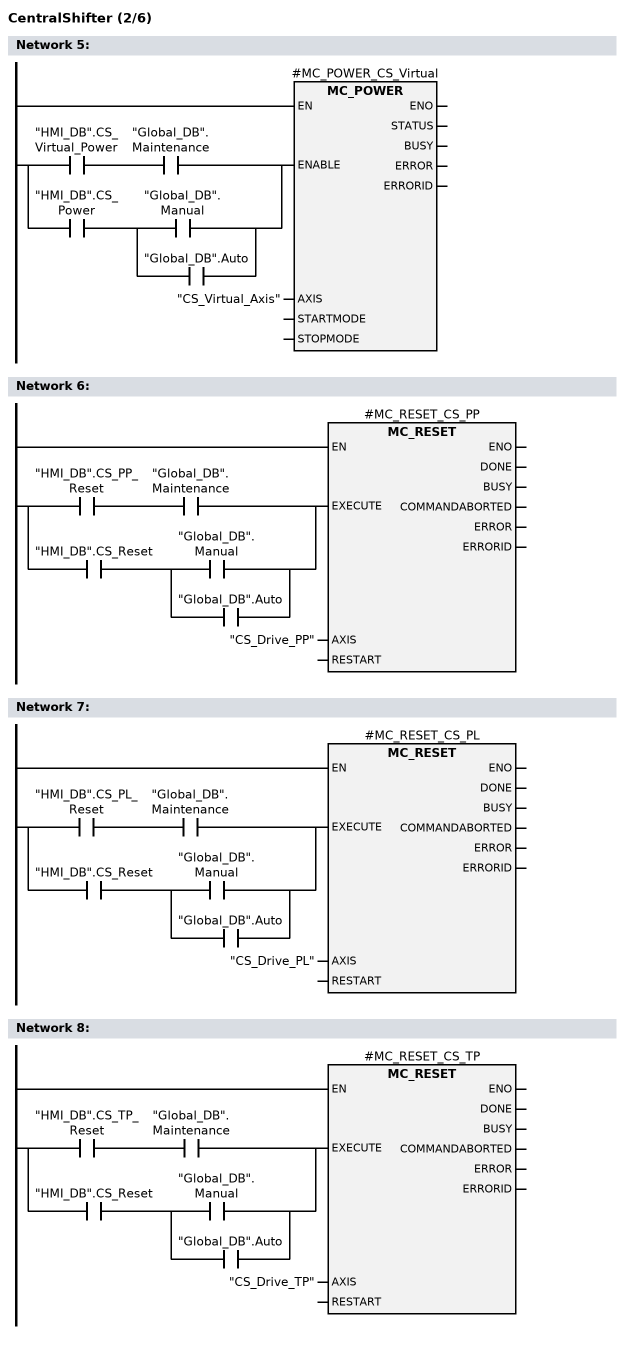
   RUNG wire#powerrail
      #MC_POWER_CS_Virtual.MC_POWER(Enable := wire#w2, Axis := "CS_Virtual_Axis", StartMode :=, StopMode :=, Status =>, Busy =>, Error =>, ErrorId =>)
   END_RUNG
   RUNG wire#powerrail
      Contact( "HMI_DB".CS_Virtual_Power )
      Contact( "Global_DB".Maintenance )
   END_RUNG wire#w2
   RUNG wire#powerrail
      Contact( "HMI_DB".CS_Power )
      wire#w1
      Contact( "Global_DB".Manual )
   END_RUNG wire#w2
   RUNG wire#w1
      Contact( "Global_DB".Auto )
   END_RUNG wire#w2
   // the same network as SCL:
   #MC_POWER_CS_Virtual(Enable := ("HMI_DB".CS_Virtual_Power AND "Global_DB".Maintenance) OR ("HMI_DB".CS_Power AND ("Global_DB".Manual OR "Global_DB".Auto)),   // MC_POWER
                        Axis := "CS_Virtual_Axis");
END_REGION

REGION Network 6
   RUNG wire#powerrail
      #MC_RESET_CS_PP.MC_RESET(Execute := wire#w2, Axis := "CS_Drive_PP", Restart :=, Done =>, Busy =>, CommandAborted =>, Error =>, ErrorId =>)
   END_RUNG
   RUNG wire#powerrail
      Contact( "HMI_DB".CS_PP_Reset )
      Contact( "Global_DB".Maintenance )
   END_RUNG wire#w2
   RUNG wire#powerrail
      Contact( "HMI_DB".CS_Reset )
      wire#w1
      Contact( "Global_DB".Manual )
   END_RUNG wire#w2
   RUNG wire#w1
      Contact( "Global_DB".Auto )
   END_RUNG wire#w2
   // the same network as SCL:
   #MC_RESET_CS_PP(Execute := ("HMI_DB".CS_PP_Reset AND "Global_DB".Maintenance) OR ("HMI_DB".CS_Reset AND ("Global_DB".Manual OR "Global_DB".Auto)),   // MC_RESET
                   Axis := "CS_Drive_PP");
END_REGION

REGION Network 7
   RUNG wire#powerrail
      #MC_RESET_CS_PL.MC_RESET(Execute := wire#w2, Axis := "CS_Drive_PL", Restart :=, Done =>, Busy =>, CommandAborted =>, Error =>, ErrorId =>)
   END_RUNG
   RUNG wire#powerrail
      Contact( "HMI_DB".CS_PL_Reset )
      Contact( "Global_DB".Maintenance )
   END_RUNG wire#w2
   RUNG wire#powerrail
      Contact( "HMI_DB".CS_Reset )
      wire#w1
      Contact( "Global_DB".Manual )
   END_RUNG wire#w2
   RUNG wire#w1
      Contact( "Global_DB".Auto )
   END_RUNG wire#w2
   // the same network as SCL:
   #MC_RESET_CS_PL(Execute := ("HMI_DB".CS_PL_Reset AND "Global_DB".Maintenance) OR ("HMI_DB".CS_Reset AND ("Global_DB".Manual OR "Global_DB".Auto)),   // MC_RESET
                   Axis := "CS_Drive_PL");
END_REGION

REGION Network 8
   RUNG wire#powerrail
      #MC_RESET_CS_TP.MC_RESET(Execute := wire#w2, Axis := "CS_Drive_TP", Restart :=, Done =>, Busy =>, CommandAborted =>, Error =>, ErrorId =>)
   END_RUNG
   RUNG wire#powerrail
      Contact( "HMI_DB".CS_TP_Reset )
      Contact( "Global_DB".Maintenance )
   END_RUNG wire#w2
   RUNG wire#powerrail
      Contact( "HMI_DB".CS_Reset )
      wire#w1
      Contact( "Global_DB".Manual )
   END_RUNG wire#w2
   RUNG wire#w1
      Contact( "Global_DB".Auto )
   END_RUNG wire#w2
   // the same network as SCL:
   #MC_RESET_CS_TP(Execute := ("HMI_DB".CS_TP_Reset AND "Global_DB".Maintenance) OR ("HMI_DB".CS_Reset AND ("Global_DB".Manual OR "Global_DB".Auto)),   // MC_RESET
                   Axis := "CS_Drive_TP");
END_REGION

REGION Network 9
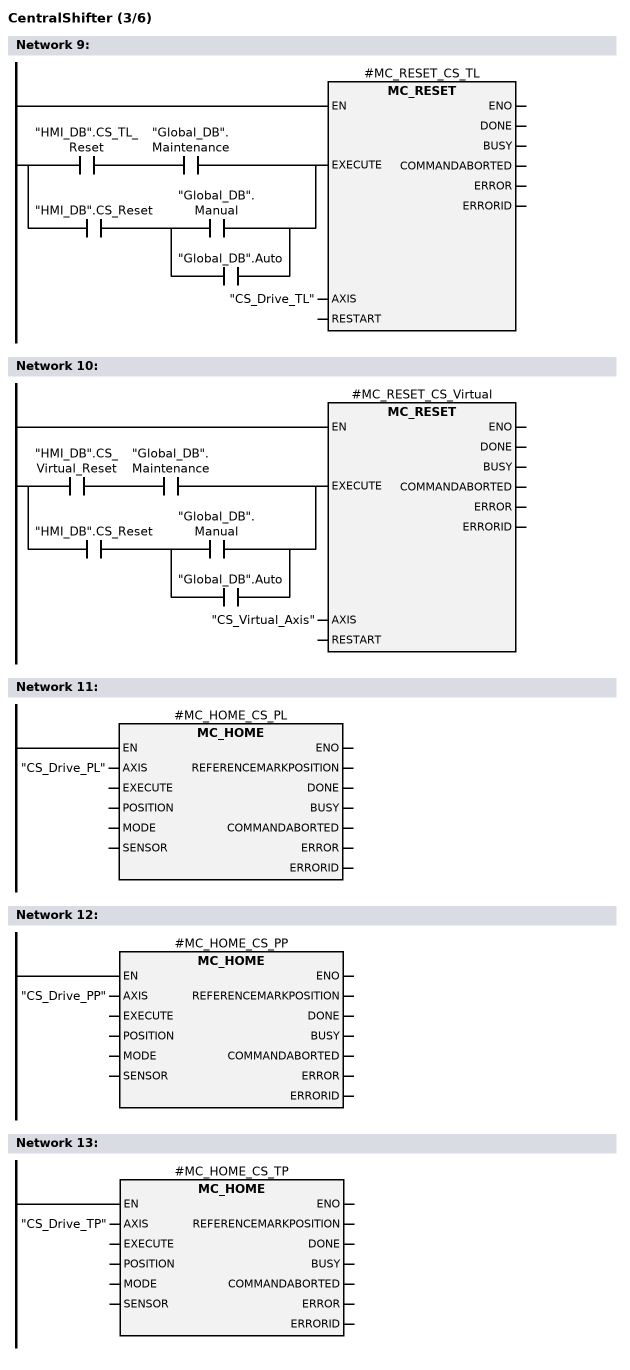
   RUNG wire#powerrail
      #MC_RESET_CS_TL.MC_RESET(Execute := wire#w2, Axis := "CS_Drive_TL", Restart :=, Done =>, Busy =>, CommandAborted =>, Error =>, ErrorId =>)
   END_RUNG
   RUNG wire#powerrail
      Contact( "HMI_DB".CS_TL_Reset )
      Contact( "Global_DB".Maintenance )
   END_RUNG wire#w2
   RUNG wire#powerrail
      Contact( "HMI_DB".CS_Reset )
      wire#w1
      Contact( "Global_DB".Manual )
   END_RUNG wire#w2
   RUNG wire#w1
      Contact( "Global_DB".Auto )
   END_RUNG wire#w2
   // the same network as SCL:
   #MC_RESET_CS_TL(Execute := ("HMI_DB".CS_TL_Reset AND "Global_DB".Maintenance) OR ("HMI_DB".CS_Reset AND ("Global_DB".Manual OR "Global_DB".Auto)),   // MC_RESET
                   Axis := "CS_Drive_TL");
END_REGION

REGION Network 10
   RUNG wire#powerrail
      #MC_RESET_CS_Virtual.MC_RESET(Execute := wire#w2, Axis := "CS_Virtual_Axis", Restart :=, Done =>, Busy =>, CommandAborted =>, Error =>, ErrorId =>)
   END_RUNG
   RUNG wire#powerrail
      Contact( "HMI_DB".CS_Virtual_Reset )
      Contact( "Global_DB".Maintenance )
   END_RUNG wire#w2
   RUNG wire#powerrail
      Contact( "HMI_DB".CS_Reset )
      wire#w1
      Contact( "Global_DB".Manual )
   END_RUNG wire#w2
   RUNG wire#w1
      Contact( "Global_DB".Auto )
   END_RUNG wire#w2
   // the same network as SCL:
   #MC_RESET_CS_Virtual(Execute := ("HMI_DB".CS_Virtual_Reset AND "Global_DB".Maintenance) OR ("HMI_DB".CS_Reset AND ("Global_DB".Manual OR "Global_DB".Auto)),   // MC_RESET
                        Axis := "CS_Virtual_Axis");
END_REGION

REGION Network 11
   RUNG wire#powerrail
      #MC_HOME_CS_PL.MC_HOME(Axis := "CS_Drive_PL", Execute :=, Position :=, Mode :=, Sensor :=, ReferenceMarkPosition =>, Done =>, Busy =>, CommandAborted =>, Error =>, ErrorId =>)
   END_RUNG
   // the same network as SCL:
   #MC_HOME_CS_PL(Axis := "CS_Drive_PL");   // MC_HOME
END_REGION

REGION Network 12
   RUNG wire#powerrail
      #MC_HOME_CS_PP.MC_HOME(Axis := "CS_Drive_PP", Execute :=, Position :=, Mode :=, Sensor :=, ReferenceMarkPosition =>, Done =>, Busy =>, CommandAborted =>, Error =>, ErrorId =>)
   END_RUNG
   // the same network as SCL:
   #MC_HOME_CS_PP(Axis := "CS_Drive_PP");   // MC_HOME
END_REGION

REGION Network 13
   RUNG wire#powerrail
      #MC_HOME_CS_TP.MC_HOME(Axis := "CS_Drive_TP", Execute :=, Position :=, Mode :=, Sensor :=, ReferenceMarkPosition =>, Done =>, Busy =>, CommandAborted =>, Error =>, ErrorId =>)
   END_RUNG
   // the same network as SCL:
   #MC_HOME_CS_TP(Axis := "CS_Drive_TP");   // MC_HOME
END_REGION

REGION Network 14
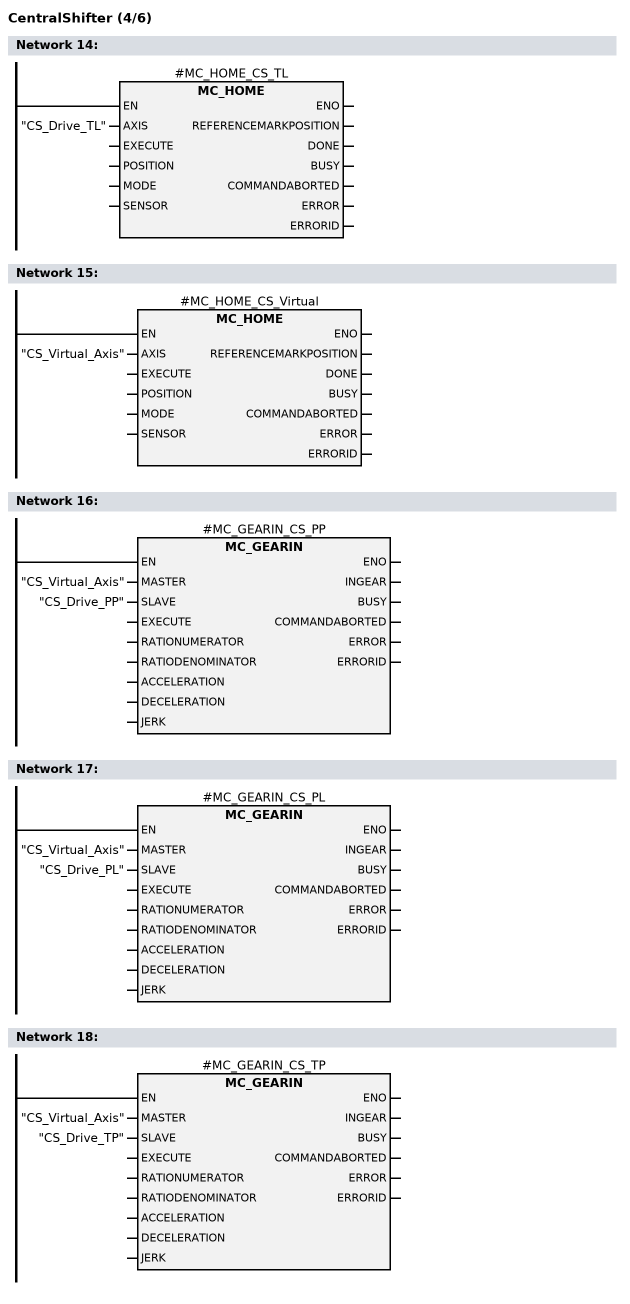
   RUNG wire#powerrail
      #MC_HOME_CS_TL.MC_HOME(Axis := "CS_Drive_TL", Execute :=, Position :=, Mode :=, Sensor :=, ReferenceMarkPosition =>, Done =>, Busy =>, CommandAborted =>, Error =>, ErrorId =>)
   END_RUNG
   // the same network as SCL:
   #MC_HOME_CS_TL(Axis := "CS_Drive_TL");   // MC_HOME
END_REGION

REGION Network 15
   RUNG wire#powerrail
      #MC_HOME_CS_Virtual.MC_HOME(Axis := "CS_Virtual_Axis", Execute :=, Position :=, Mode :=, Sensor :=, ReferenceMarkPosition =>, Done =>, Busy =>, CommandAborted =>, Error =>, ErrorId =>)
   END_RUNG
   // the same network as SCL:
   #MC_HOME_CS_Virtual(Axis := "CS_Virtual_Axis");   // MC_HOME
END_REGION

REGION Network 16
   RUNG wire#powerrail
      #MC_GEARIN_CS_PP.MC_GEARIN(Master := "CS_Virtual_Axis", Slave := "CS_Drive_PP", Execute :=, RatioNumerator :=, RatioDenominator :=, Acceleration :=, Deceleration :=, Jerk :=, InGear =>, Busy =>, CommandAborted =>, Error =>, ErrorId =>)
   END_RUNG
   // the same network as SCL:
   #MC_GEARIN_CS_PP(Master := "CS_Virtual_Axis", Slave := "CS_Drive_PP");   // MC_GEARIN
END_REGION

REGION Network 17
   RUNG wire#powerrail
      #MC_GEARIN_CS_PL.MC_GEARIN(Master := "CS_Virtual_Axis", Slave := "CS_Drive_PL", Execute :=, RatioNumerator :=, RatioDenominator :=, Acceleration :=, Deceleration :=, Jerk :=, InGear =>, Busy =>, CommandAborted =>, Error =>, ErrorId =>)
   END_RUNG
   // the same network as SCL:
   #MC_GEARIN_CS_PL(Master := "CS_Virtual_Axis", Slave := "CS_Drive_PL");   // MC_GEARIN
END_REGION

REGION Network 18
   RUNG wire#powerrail
      #MC_GEARIN_CS_TP.MC_GEARIN(Master := "CS_Virtual_Axis", Slave := "CS_Drive_TP", Execute :=, RatioNumerator :=, RatioDenominator :=, Acceleration :=, Deceleration :=, Jerk :=, InGear =>, Busy =>, CommandAborted =>, Error =>, ErrorId =>)
   END_RUNG
   // the same network as SCL:
   #MC_GEARIN_CS_TP(Master := "CS_Virtual_Axis", Slave := "CS_Drive_TP");   // MC_GEARIN
END_REGION

REGION Network 19
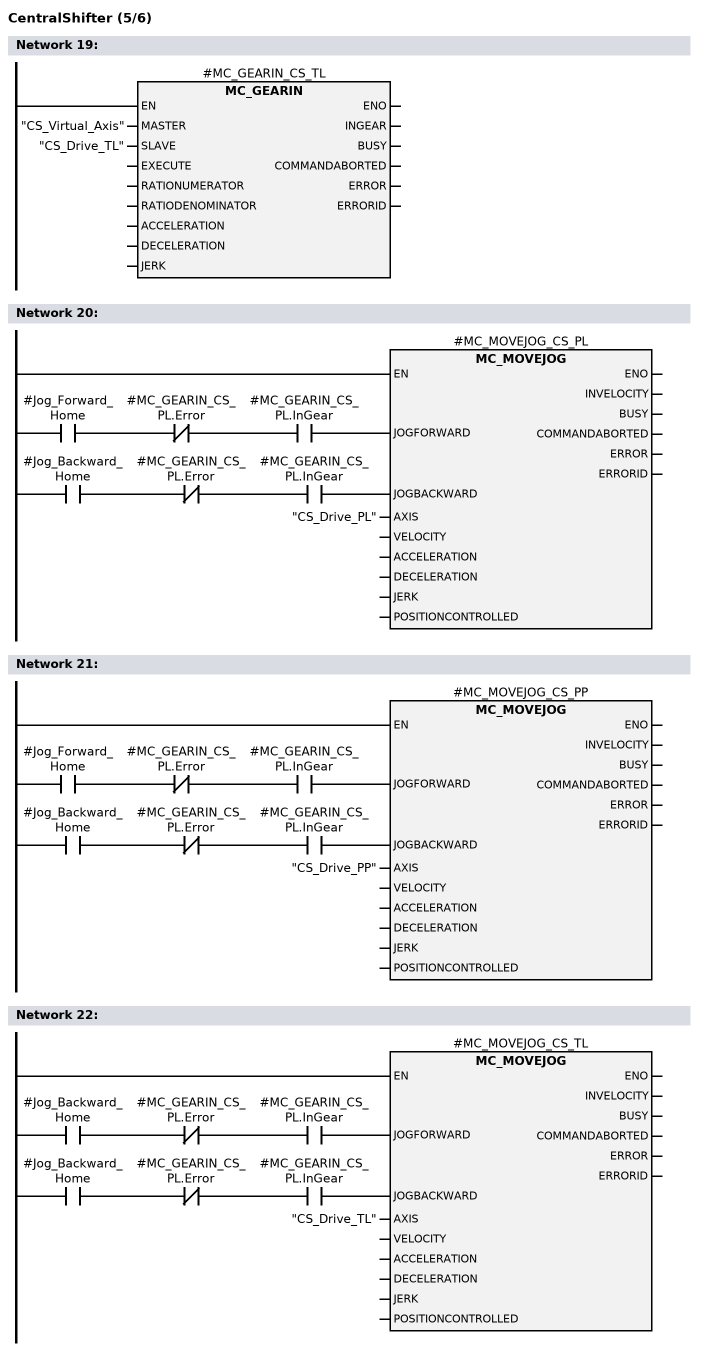
   RUNG wire#powerrail
      #MC_GEARIN_CS_TL.MC_GEARIN(Master := "CS_Virtual_Axis", Slave := "CS_Drive_TL", Execute :=, RatioNumerator :=, RatioDenominator :=, Acceleration :=, Deceleration :=, Jerk :=, InGear =>, Busy =>, CommandAborted =>, Error =>, ErrorId =>)
   END_RUNG
   // the same network as SCL:
   #MC_GEARIN_CS_TL(Master := "CS_Virtual_Axis", Slave := "CS_Drive_TL");   // MC_GEARIN
END_REGION

REGION Network 20
   RUNG wire#powerrail
      #MC_MOVEJOG_CS_PL.MC_MOVEJOG(JogForward := wire#w1, JogBackward := wire#w2, Axis := "CS_Drive_PL", Velocity :=, Acceleration :=, Deceleration :=, Jerk :=, PositionControlled :=, InVelocity =>, Busy =>, CommandAborted =>, Error =>, ErrorId =>)
   END_RUNG
   RUNG wire#powerrail
      Contact( #Jog_Forward_Home )
      I_Contact( #MC_GEARIN_CS_PL.Error )
      Contact( #MC_GEARIN_CS_PL.InGear )
   END_RUNG wire#w1
   RUNG wire#powerrail
      Contact( #Jog_Backward_Home )
      I_Contact( #MC_GEARIN_CS_PL.Error )
      Contact( #MC_GEARIN_CS_PL.InGear )
   END_RUNG wire#w2
   // the same network as SCL:
   #MC_MOVEJOG_CS_PL(JogForward := #Jog_Forward_Home AND NOT #MC_GEARIN_CS_PL.Error AND #MC_GEARIN_CS_PL.InGear,   // MC_MOVEJOG
                     JogBackward := #Jog_Backward_Home AND NOT #MC_GEARIN_CS_PL.Error AND #MC_GEARIN_CS_PL.InGear,
                     Axis := "CS_Drive_PL");
END_REGION

REGION Network 21
   RUNG wire#powerrail
      #MC_MOVEJOG_CS_PP.MC_MOVEJOG(JogForward := wire#w1, JogBackward := wire#w2, Axis := "CS_Drive_PP", Velocity :=, Acceleration :=, Deceleration :=, Jerk :=, PositionControlled :=, InVelocity =>, Busy =>, CommandAborted =>, Error =>, ErrorId =>)
   END_RUNG
   RUNG wire#powerrail
      Contact( #Jog_Forward_Home )
      I_Contact( #MC_GEARIN_CS_PL.Error )
      Contact( #MC_GEARIN_CS_PL.InGear )
   END_RUNG wire#w1
   RUNG wire#powerrail
      Contact( #Jog_Backward_Home )
      I_Contact( #MC_GEARIN_CS_PL.Error )
      Contact( #MC_GEARIN_CS_PL.InGear )
   END_RUNG wire#w2
   // the same network as SCL:
   #MC_MOVEJOG_CS_PP(JogForward := #Jog_Forward_Home AND NOT #MC_GEARIN_CS_PL.Error AND #MC_GEARIN_CS_PL.InGear,   // MC_MOVEJOG
                     JogBackward := #Jog_Backward_Home AND NOT #MC_GEARIN_CS_PL.Error AND #MC_GEARIN_CS_PL.InGear,
                     Axis := "CS_Drive_PP");
END_REGION

REGION Network 22
   RUNG wire#powerrail
      #MC_MOVEJOG_CS_TL.MC_MOVEJOG(JogForward := wire#w1, JogBackward := wire#w2, Axis := "CS_Drive_TL", Velocity :=, Acceleration :=, Deceleration :=, Jerk :=, PositionControlled :=, InVelocity =>, Busy =>, CommandAborted =>, Error =>, ErrorId =>)
   END_RUNG
   RUNG wire#powerrail
      Contact( #Jog_Backward_Home )
      I_Contact( #MC_GEARIN_CS_PL.Error )
      Contact( #MC_GEARIN_CS_PL.InGear )
   END_RUNG wire#w1
   RUNG wire#powerrail
      Contact( #Jog_Backward_Home )
      I_Contact( #MC_GEARIN_CS_PL.Error )
      Contact( #MC_GEARIN_CS_PL.InGear )
   END_RUNG wire#w2
   // the same network as SCL:
   #MC_MOVEJOG_CS_TL(JogForward := #Jog_Backward_Home AND NOT #MC_GEARIN_CS_PL.Error AND #MC_GEARIN_CS_PL.InGear,   // MC_MOVEJOG
                     JogBackward := #Jog_Backward_Home AND NOT #MC_GEARIN_CS_PL.Error AND #MC_GEARIN_CS_PL.InGear,
                     Axis := "CS_Drive_TL");
END_REGION

REGION Network 23
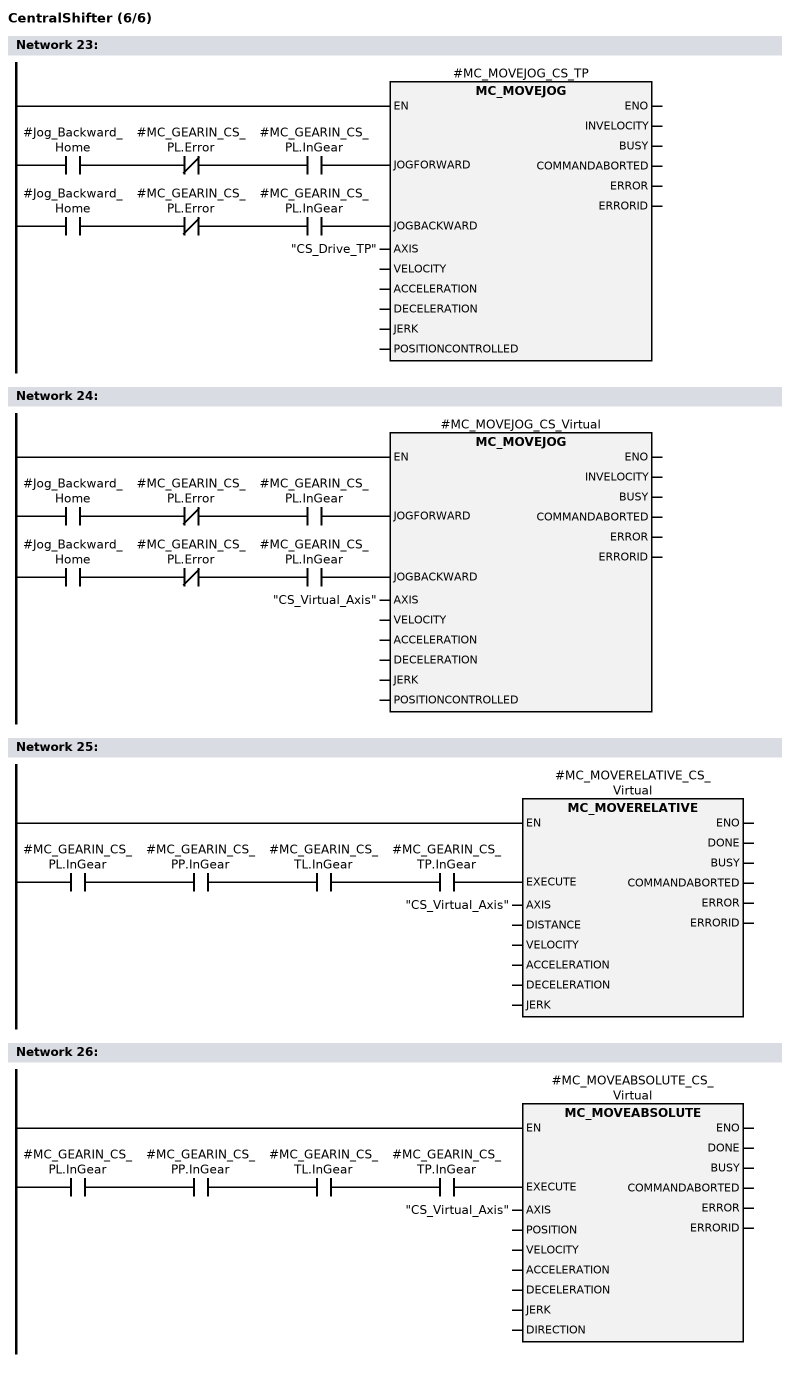
   RUNG wire#powerrail
      #MC_MOVEJOG_CS_TP.MC_MOVEJOG(JogForward := wire#w1, JogBackward := wire#w2, Axis := "CS_Drive_TP", Velocity :=, Acceleration :=, Deceleration :=, Jerk :=, PositionControlled :=, InVelocity =>, Busy =>, CommandAborted =>, Error =>, ErrorId =>)
   END_RUNG
   RUNG wire#powerrail
      Contact( #Jog_Backward_Home )
      I_Contact( #MC_GEARIN_CS_PL.Error )
      Contact( #MC_GEARIN_CS_PL.InGear )
   END_RUNG wire#w1
   RUNG wire#powerrail
      Contact( #Jog_Backward_Home )
      I_Contact( #MC_GEARIN_CS_PL.Error )
      Contact( #MC_GEARIN_CS_PL.InGear )
   END_RUNG wire#w2
   // the same network as SCL:
   #MC_MOVEJOG_CS_TP(JogForward := #Jog_Backward_Home AND NOT #MC_GEARIN_CS_PL.Error AND #MC_GEARIN_CS_PL.InGear,   // MC_MOVEJOG
                     JogBackward := #Jog_Backward_Home AND NOT #MC_GEARIN_CS_PL.Error AND #MC_GEARIN_CS_PL.InGear,
                     Axis := "CS_Drive_TP");
END_REGION

REGION Network 24
   RUNG wire#powerrail
      #MC_MOVEJOG_CS_Virtual.MC_MOVEJOG(JogForward := wire#w1, JogBackward := wire#w2, Axis := "CS_Virtual_Axis", Velocity :=, Acceleration :=, Deceleration :=, Jerk :=, PositionControlled :=, InVelocity =>, Busy =>, CommandAborted =>, Error =>, ErrorId =>)
   END_RUNG
   RUNG wire#powerrail
      Contact( #Jog_Backward_Home )
      I_Contact( #MC_GEARIN_CS_PL.Error )
      Contact( #MC_GEARIN_CS_PL.InGear )
   END_RUNG wire#w1
   RUNG wire#powerrail
      Contact( #Jog_Backward_Home )
      I_Contact( #MC_GEARIN_CS_PL.Error )
      Contact( #MC_GEARIN_CS_PL.InGear )
   END_RUNG wire#w2
   // the same network as SCL:
   #MC_MOVEJOG_CS_Virtual(JogForward := #Jog_Backward_Home AND NOT #MC_GEARIN_CS_PL.Error AND #MC_GEARIN_CS_PL.InGear,   // MC_MOVEJOG
                          JogBackward := #Jog_Backward_Home AND NOT #MC_GEARIN_CS_PL.Error AND #MC_GEARIN_CS_PL.InGear,
                          Axis := "CS_Virtual_Axis");
END_REGION

REGION Network 25
   RUNG wire#powerrail
      #MC_MOVERELATIVE_CS_Virtual.MC_MOVERELATIVE(Execute := wire#w1, Axis := "CS_Virtual_Axis", Distance :=, Velocity :=, Acceleration :=, Deceleration :=, Jerk :=, Done =>, Busy =>, CommandAborted =>, Error =>, ErrorId =>)
   END_RUNG
   RUNG wire#powerrail
      Contact( #MC_GEARIN_CS_PL.InGear )
      Contact( #MC_GEARIN_CS_PP.InGear )
      Contact( #MC_GEARIN_CS_TL.InGear )
      Contact( #MC_GEARIN_CS_TP.InGear )
   END_RUNG wire#w1
   // the same network as SCL:
   #MC_MOVERELATIVE_CS_Virtual(Execute := #MC_GEARIN_CS_PL.InGear AND #MC_GEARIN_CS_PP.InGear AND #MC_GEARIN_CS_TL.InGear AND #MC_GEARIN_CS_TP.InGear,   // MC_MOVERELATIVE
                           Axis := "CS_Virtual_Axis");
END_REGION

REGION Network 26
   RUNG wire#powerrail
      #MC_MOVEABSOLUTE_CS_Virtual.MC_MOVEABSOLUTE(Execute := wire#w1, Axis := "CS_Virtual_Axis", Position :=, Velocity :=, Acceleration :=, Deceleration :=, Jerk :=, Direction :=, Done =>, Busy =>, CommandAborted =>, Error =>, ErrorId =>)
   END_RUNG
   RUNG wire#powerrail
      Contact( #MC_GEARIN_CS_PL.InGear )
      Contact( #MC_GEARIN_CS_PP.InGear )
      Contact( #MC_GEARIN_CS_TL.InGear )
      Contact( #MC_GEARIN_CS_TP.InGear )
   END_RUNG wire#w1
   // the same network as SCL:
   #MC_MOVEABSOLUTE_CS_Virtual(Execute := #MC_GEARIN_CS_PL.InGear AND #MC_GEARIN_CS_PP.InGear AND #MC_GEARIN_CS_TL.InGear AND #MC_GEARIN_CS_TP.InGear,   // MC_MOVEABSOLUTE
                           Axis := "CS_Virtual_Axis");
END_REGION

REGION Network 27 (SCL): Homing
   IF "HMI_DB".CS_Homing AND NOT "iCS_SensorHoming_Left" AND (#Homeing_Status = 0 OR #Homeing_Status = 5) THEN
       #Jog_Backward_Home := 1;
       #Jog_Forward_Home := 0;
       #Jog_Velocity := 15;
       #Homeing_Status := 1;

   ELSIF "HMI_DB".CS_Homing  AND "iCS_SensorHoming_Left" THEN
       #Jog_Backward_Home := 0;
       #Jog_Forward_Home := 1;
       #Jog_Velocity := 1;
       #Homeing_Status := 2;

   ELSIF "HMI_DB".CS_Homing  AND NOT "iCS_SensorHoming_Left" AND #Homeing_Status = 2 THEN
       #Jog_Backward_Home := 0;
       #Jog_Forward_Home := 0;
       #Homeing_Status := 3;

   ELSIF "HMI_DB".CS_Homing AND NOT "iCS_SensorHoming_Left" AND #Homeing_Status = 3 THEN
       #MC_HOME_CS_PL.Execute := 1;
       #MC_HOME_CS_PP.Execute := 1;
       #MC_HOME_CS_TP.Execute := 1;
       #MC_HOME_CS_TL.Execute := 1;
       #MC_HOME_CS_Virtual.Execute := 1;
       #Homeing_Status := 4;
       "HMI_DB".CS_Homing := 0;

   ELSIF #Homeing_Status = 4 AND #MC_HOME_CS_PL.Done AND #MC_HOME_CS_PL.Done AND #MC_HOME_CS_TL.Done AND #MC_HOME_CS_TL.Done AND #MC_HOME_CS_Virtual.Done AND "CS_Virtual_Axis".Position <= 1 THEN
       #MC_HOME_CS_PL.Execute := 0;
       #MC_HOME_CS_PP.Execute := 0;
       #MC_HOME_CS_TP.Execute := 0;
       #MC_HOME_CS_TL.Execute := 0;
       #Homeing_Status := 5; //ready
       "HMI_DB".CS_Homing := 0;

   ELSIF #Homeing_Status = 5 THEN
       "HMI_DB".CS_Homing := 0;
       IF "CS_Virtual_Axis".Position >= 1 THEN
           #Homeing_Status := 0;

       END_IF;
   END_IF;
END_REGION
END_FUNCTION_BLOCK

FUNCTION_BLOCK "Main_Safety_RTG1"   // FB1, F_FBD
{ S7_Optimized_Access := 'TRUE' }
// stored: AutoNumber false
BEGIN
END_FUNCTION_BLOCK

FUNCTION_BLOCK "SideShifter_Hydraulic"   // FB4, LAD
{ S7_Optimized_Access := 'TRUE' }
// stored: MemoryReserve 100, SetENOAutomatically false
   VAR_INPUT
      Actuators_Down : Bool;
      Actuators_Up : Bool;
      Hydraulic_Unit : Bool;
      iAct1_1_Sensor_Up : Bool;
      iAct1_1_Sensor_Down : Bool;
      iAct1_2_Sensor_Up : Bool;
      iAct1_2_Sensor_Down : Bool;
   END_VAR
   VAR_OUTPUT
      oValve1_Up : Bool;
      oValve1_Down : Bool;
      oHydraulic_Unit : Bool;
   END_VAR
BEGIN

REGION Network 1
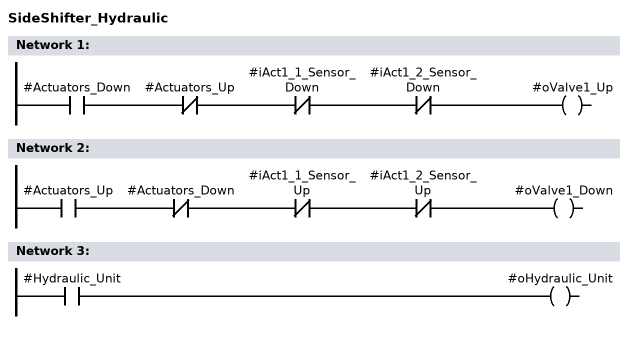
   RUNG wire#powerrail
      Contact( #Actuators_Down )
      I_Contact( #Actuators_Up )
      I_Contact( #iAct1_1_Sensor_Down )
      I_Contact( #iAct1_2_Sensor_Down )
      Coil( #oValve1_Up )
   END_RUNG
   // the same network as SCL:
   #oValve1_Up := #Actuators_Down AND NOT #Actuators_Up AND NOT #iAct1_1_Sensor_Down AND NOT #iAct1_2_Sensor_Down;
END_REGION

REGION Network 2
   RUNG wire#powerrail
      Contact( #Actuators_Up )
      I_Contact( #Actuators_Down )
      I_Contact( #iAct1_1_Sensor_Up )
      I_Contact( #iAct1_2_Sensor_Up )
      Coil( #oValve1_Down )
   END_RUNG
   // the same network as SCL:
   #oValve1_Down := #Actuators_Up AND NOT #Actuators_Down AND NOT #iAct1_1_Sensor_Up AND NOT #iAct1_2_Sensor_Up;
END_REGION

REGION Network 3
   RUNG wire#powerrail
      Contact( #Hydraulic_Unit )
      Coil( #oHydraulic_Unit )
   END_RUNG
   // the same network as SCL:
   #oHydraulic_Unit := #Hydraulic_Unit;
END_REGION
END_FUNCTION_BLOCK

FUNCTION_BLOCK "Initialisation"
{ S7_Optimized_Access := 'TRUE' }
VERSION : 0.1
   VAR_TEMP 
      i : Int;
      j : Int;
   END_VAR


BEGIN
	REGION Stations_Sensors
	    
	    // row 1
	    
	    "Pallets_Stations".Stations[1, 1].SensorA := "Sz5_ST35_SenA";
	    "Pallets_Stations".Stations[1, 1].SensorB := "Sz5_ST35_SenB";
	    "Pallets_Stations".Stations[1, 1].SensorC := "Sz5_ST35_SenC";
	    "Pallets_Stations".Stations[1, 1].SensorD := "Sz5_ST35_SenD";
	    
	    "Pallets_Stations".Stations[1, 2].SensorA := "Sz5_ST34_SenA";
	    "Pallets_Stations".Stations[1, 2].SensorB := "Sz5_ST34_SenB";
	    "Pallets_Stations".Stations[1, 2].SensorC := "Sz5_ST34_SenC";
	    "Pallets_Stations".Stations[1, 2].SensorD := "Sz5_ST34_SenD";
	    
	    "Pallets_Stations".Stations[1, 3].SensorA := "Sz4_ST33_SenA";
	    "Pallets_Stations".Stations[1, 3].SensorB := "Sz4_ST33_SenB";
	    "Pallets_Stations".Stations[1, 3].SensorC := "Sz4_ST33_SenC";
	    "Pallets_Stations".Stations[1, 3].SensorD := "Sz4_ST33_SenD";
	    
	    "Pallets_Stations".Stations[1, 4].SensorA := "Sz4_ST32_SenA";
	    "Pallets_Stations".Stations[1, 4].SensorB := "Sz4_ST32_SenB";
	    "Pallets_Stations".Stations[1, 4].SensorC := "Sz4_ST32_SenC";
	    "Pallets_Stations".Stations[1, 4].SensorD := "Sz4_ST32_SenD";
	    
	    "Pallets_Stations".Stations[1, 5].SensorA := "Sz3_ST31_SenA";
	    "Pallets_Stations".Stations[1, 5].SensorB := "Sz3_ST31_SenB";
	    "Pallets_Stations".Stations[1, 5].SensorC := "Sz3_ST31_SenC";
	    "Pallets_Stations".Stations[1, 5].SensorD := "Sz3_ST31_SenD";
	    
	    "Pallets_Stations".Stations[1, 6].SensorA := "Sz3_ST30_SenA";
	    "Pallets_Stations".Stations[1, 6].SensorB := "Sz3_ST30_SenB";
	    "Pallets_Stations".Stations[1, 6].SensorC := "Sz3_ST30_SenC";
	    "Pallets_Stations".Stations[1, 6].SensorD := "Sz3_ST30_SenD";
	    
	    "Pallets_Stations".Stations[1, 7].SensorA := "Sz3_ST29_SenA";
	    "Pallets_Stations".Stations[1, 7].SensorB := "Sz3_ST29_SenB";
	    "Pallets_Stations".Stations[1, 7].SensorC := "Sz3_ST29_SenC";
	    "Pallets_Stations".Stations[1, 7].SensorD := "Sz3_ST29_SenD";
	    
	    "Pallets_Stations".Stations[1, 8].SensorA := "Sz2_ST28_SenA";
	    "Pallets_Stations".Stations[1, 8].SensorB := "Sz2_ST28_SenB";
	    "Pallets_Stations".Stations[1, 8].SensorC := "Sz2_ST28_SenC";
	    "Pallets_Stations".Stations[1, 8].SensorD := "Sz2_ST28_SenD";
	    
	    "Pallets_Stations".Stations[1, 9].SensorA := "Sz2_ST27_SenA";
	    "Pallets_Stations".Stations[1, 9].SensorB := "Sz2_ST27_SenB";
	    "Pallets_Stations".Stations[1, 9].SensorC := "Sz2_ST27_SenC";
	    "Pallets_Stations".Stations[1, 9].SensorD := "Sz2_ST27_SenD";
	    
	    "Pallets_Stations".Stations[1, 10].SensorA := "Sz1_St26_SenA";
	    "Pallets_Stations".Stations[1, 10].SensorB := "Sz1_St26_SenB";
	    "Pallets_Stations".Stations[1, 10].SensorC := "Sz1_St26_SenC";
	    "Pallets_Stations".Stations[1, 10].SensorD := "Sz1_St26_SenD";
	    
	    "Pallets_Stations".Stations[1, 11].SensorA := "Sz1_St25_SenA";
	    "Pallets_Stations".Stations[1, 11].SensorB := "Sz1_St25_SenB";
	    "Pallets_Stations".Stations[1, 11].SensorC := "Sz1_St25_SenC";
	    "Pallets_Stations".Stations[1, 11].SensorD := "Sz1_St25_SenD";
	    
	    //row 2
	    
	    "Pallets_Stations".Stations[2, 1].SensorA := "Sz5_ST01_SenA";
	    "Pallets_Stations".Stations[2, 1].SensorB := "Sz5_ST01_SenB";
	    "Pallets_Stations".Stations[2, 1].SensorC := "Sz5_ST01_SenC";
	    "Pallets_Stations".Stations[2, 1].SensorD := "Sz5_ST01_SenD";
	    
	    "Pallets_Stations".Stations[2, 2].SensorA := "Sz5_ST02_SenA";
	    "Pallets_Stations".Stations[2, 2].SensorB := "Sz5_ST02_SenB";
	    "Pallets_Stations".Stations[2, 2].SensorC := "Sz5_ST02_SenC";
	    "Pallets_Stations".Stations[2, 2].SensorD := "Sz5_ST02_SenD";
	    
	    "Pallets_Stations".Stations[2, 3].SensorA := "Sz5_ST38_SenA";
	    "Pallets_Stations".Stations[2, 3].SensorB := "Sz5_ST38_SenB";
	    "Pallets_Stations".Stations[2, 3].SensorC := "Sz5_ST38_SenC";
	    "Pallets_Stations".Stations[2, 3].SensorD := "Sz5_ST38_SenD";
	    
	    "Pallets_Stations".Stations[2, 4].SensorA := "Sz4_ST36_SenA";
	    "Pallets_Stations".Stations[2, 4].SensorB := "Sz4_ST36_SenB";
	    "Pallets_Stations".Stations[2, 4].SensorC := "Sz4_ST36_SenC";
	    "Pallets_Stations".Stations[2, 4].SensorD := "Sz4_ST36_SenD";
	    
	    "Pallets_Stations".Stations[2, 5].SensorA := "Sz4_ST37_SenA";
	    "Pallets_Stations".Stations[2, 5].SensorB := "Sz4_ST37_SenB";
	    "Pallets_Stations".Stations[2, 5].SensorC := "Sz4_ST37_SenC";
	    "Pallets_Stations".Stations[2, 5].SensorD := "Sz4_ST37_SenD";
	    
	    "Pallets_Stations".Stations[2, 6].SensorA := "Sz3_ST18_SenA";
	    "Pallets_Stations".Stations[2, 6].SensorB := "Sz3_ST18_SenB";
	    "Pallets_Stations".Stations[2, 6].SensorC := "Sz3_ST18_SenC";
	    "Pallets_Stations".Stations[2, 6].SensorD := "Sz3_ST18_SenD";
	    
	    "Pallets_Stations".Stations[2, 7].SensorA := "Sz3_ST19_SenA";
	    "Pallets_Stations".Stations[2, 7].SensorB := "Sz3_ST19_SenB";
	    "Pallets_Stations".Stations[2, 7].SensorC := "Sz3_ST19_SenC";
	    "Pallets_Stations".Stations[2, 7].SensorD := "Sz3_ST19_SenD";
	    
	    "Pallets_Stations".Stations[2, 8].SensorA := "Sz3_ST20_SenA";
	    "Pallets_Stations".Stations[2, 8].SensorB := "Sz3_ST20_SenB";
	    "Pallets_Stations".Stations[2, 8].SensorC := "Sz3_ST20_SenC";
	    "Pallets_Stations".Stations[2, 8].SensorD := "Sz3_ST20_SenD";
	    
	    "Pallets_Stations".Stations[2, 9].SensorA := "Sz2_ST21_SenA";
	    "Pallets_Stations".Stations[2, 9].SensorB := "Sz2_ST21_SenB";
	    "Pallets_Stations".Stations[2, 9].SensorC := "Sz2_ST21_SenC";
	    "Pallets_Stations".Stations[2, 9].SensorD := "Sz2_ST21_SenD";
	    
	    "Pallets_Stations".Stations[2, 10].SensorA := "Sz2_ST22_SenA";
	    "Pallets_Stations".Stations[2, 10].SensorB := "Sz2_ST22_SenB";
	    "Pallets_Stations".Stations[2, 10].SensorC := "Sz2_ST22_SenC";
	    "Pallets_Stations".Stations[2, 10].SensorD := "Sz2_ST22_SenD";
	    
	    "Pallets_Stations".Stations[2, 11].SensorA := "Sz1_St23_SenA";
	    "Pallets_Stations".Stations[2, 11].SensorB := "Sz1_St23_SenB";
	    "Pallets_Stations".Stations[2, 11].SensorC := "Sz1_St23_SenC";
	    "Pallets_Stations".Stations[2, 11].SensorD := "Sz1_St23_SenD";
	    
	    "Pallets_Stations".Stations[2, 12].SensorA := "Sz1_St24_SenA";
	    "Pallets_Stations".Stations[2, 12].SensorB := "Sz1_St24_SenB";
	    "Pallets_Stations".Stations[2, 12].SensorC := "Sz1_St24_SenC";
	    "Pallets_Stations".Stations[2, 12].SensorD := "Sz1_St24_SenD";
	    
	    // row 3
	    
	    "Pallets_Stations".Stations[3, 1].SensorA := "Sz7_ST03_SenA";
	    "Pallets_Stations".Stations[3, 1].SensorB := "Sz7_ST03_SenB";
	    "Pallets_Stations".Stations[3, 1].SensorC := "Sz7_ST03_SenC";
	    "Pallets_Stations".Stations[3, 1].SensorD := "Sz7_ST03_SenD";
	    
	    "Pallets_Stations".Stations[3, 11].SensorA := "Sz11_ST17_SenA";
	    "Pallets_Stations".Stations[3, 11].SensorB := "Sz11_ST17_SenB";
	    "Pallets_Stations".Stations[3, 11].SensorC := "Sz11_ST17_SenC";
	    "Pallets_Stations".Stations[3, 11].SensorD := "Sz11_ST17_SenD";
	    
	    // row 4
	    
	    "Pallets_Stations".Stations[4, 1].SensorA := "Sz7_ST04_SenA";
	    "Pallets_Stations".Stations[4, 1].SensorB := "Sz7_ST04_SenB";
	    "Pallets_Stations".Stations[4, 1].SensorC := "Sz7_ST04_SenC";
	    "Pallets_Stations".Stations[4, 1].SensorD := "Sz7_ST04_SenD";
	    
	    "Pallets_Stations".Stations[4, 2].SensorA := "Sz7_ST05_SenA";
	    "Pallets_Stations".Stations[4, 2].SensorB := "Sz7_ST05_SenB";
	    "Pallets_Stations".Stations[4, 2].SensorC := "Sz7_ST05_SenC";
	    "Pallets_Stations".Stations[4, 2].SensorD := "Sz7_ST05_SenD";
	   
	    "Pallets_Stations".Stations[4, 3].SensorA := "Sz8_ST06_SenA";
	    "Pallets_Stations".Stations[4, 3].SensorB := "Sz8_ST06_SenB";
	    "Pallets_Stations".Stations[4, 3].SensorC := "Sz8_ST06_SenC";
	    "Pallets_Stations".Stations[4, 3].SensorD := "Sz8_ST06_SenD";
	    
	    "Pallets_Stations".Stations[4, 4].SensorA := "Sz8_ST07_SenA";
	    "Pallets_Stations".Stations[4, 4].SensorB := "Sz8_ST07_SenB";
	    "Pallets_Stations".Stations[4, 4].SensorC := "Sz8_ST07_SenC";
	    "Pallets_Stations".Stations[4, 4].SensorD := "Sz8_ST07_SenD";
	    
	    "Pallets_Stations".Stations[4, 5].SensorA := "Sz8_ST08_SenA";
	    "Pallets_Stations".Stations[4, 5].SensorB := "Sz8_ST08_SenB";
	    "Pallets_Stations".Stations[4, 5].SensorC := "Sz8_ST08_SenC";
	    "Pallets_Stations".Stations[4, 5].SensorD := "Sz8_ST08_SenD";
	    
	    "Pallets_Stations".Stations[4, 6].SensorA := "Sz9_ST09_SenA";
	    "Pallets_Stations".Stations[4, 6].SensorB := "Sz9_ST09_SenB";
	    "Pallets_Stations".Stations[4, 6].SensorC := "Sz9_ST09_SenC";
	    "Pallets_Stations".Stations[4, 6].SensorD := "Sz9_ST09_SenD";
	    
	    "Pallets_Stations".Stations[4, 7].SensorA := "Sz9_ST10_SenA";
	    "Pallets_Stations".Stations[4, 7].SensorB := "Sz9_ST10_SenB";
	    "Pallets_Stations".Stations[4, 7].SensorC := "Sz9_ST10_SenC";
	    "Pallets_Stations".Stations[4, 7].SensorD := "Sz9_ST10_SenD";
	    
	    "Pallets_Stations".Stations[4, 8].SensorA := "Sz10_ST11_SenA";
	    "Pallets_Stations".Stations[4, 8].SensorB := "Sz10_ST11_SenB";
	    "Pallets_Stations".Stations[4, 8].SensorC := "Sz10_ST11_SenC";
	    "Pallets_Stations".Stations[4, 8].SensorD := "Sz10_ST11_SenD";
	    
	    "Pallets_Stations".Stations[4, 9].SensorA := "Sz10_ST12_SenA";
	    "Pallets_Stations".Stations[4, 9].SensorB := "Sz10_ST12_SenB";
	    "Pallets_Stations".Stations[4, 9].SensorC := "Sz10_ST12_SenC";
	    "Pallets_Stations".Stations[4, 9].SensorD := "Sz10_ST12_SenD";
	    
	    "Pallets_Stations".Stations[4, 10].SensorA := "Sz11_ST13_SenA";
	    "Pallets_Stations".Stations[4, 10].SensorB := "Sz11_ST13_SenB";
	    "Pallets_Stations".Stations[4, 10].SensorC := "Sz11_ST13_SenC";
	    "Pallets_Stations".Stations[4, 10].SensorD := "Sz11_ST13_SenD";
	    
	    "Pallets_Stations".Stations[4, 11].SensorA := "Sz11_ST14_SenA";
	    "Pallets_Stations".Stations[4, 11].SensorB := "Sz11_ST14_SenB";
	    "Pallets_Stations".Stations[4, 11].SensorC := "Sz11_ST14_SenC";
	    "Pallets_Stations".Stations[4, 11].SensorD := "Sz11_ST14_SenD";
	    
	END_REGION
	
	REGION Station_Status
	    
	    FOR #i := 1 TO 4 DO
	        FOR #j := 1 TO 12 DO
	            // CentralShifter
	            IF (#i = 3 AND (#j >= 2 AND #j <= 10)) OR
	                ((#i = 1 OR #i = 3 OR #i = 4) AND #j = 12) THEN // Last column
	                "Pallets_Stations".Stations[#i, #j].IsOccupied := TRUE;
	                "Pallets_Stations".Stations[#i, #j].IsEmpty := FALSE;
	                // All sensors are True
	            ELSIF "Pallets_Stations".Stations[#i, #j].SensorA AND
	                "Pallets_Stations".Stations[#i, #j].SensorB AND
	                "Pallets_Stations".Stations[#i, #j].SensorC AND
	                "Pallets_Stations".Stations[#i, #j].SensorD THEN
	                "Pallets_Stations".Stations[#i, #j].IsOccupied := TRUE;
	                "Pallets_Stations".Stations[#i, #j].IsEmpty := FALSE;
	                // All sensors are False
	            ELSIF NOT "Pallets_Stations".Stations[#i, #j].SensorA AND
	                NOT "Pallets_Stations".Stations[#i, #j].SensorB AND
	                NOT "Pallets_Stations".Stations[#i, #j].SensorC AND
	                NOT "Pallets_Stations".Stations[#i, #j].SensorD THEN
	                "Pallets_Stations".Stations[#i, #j].IsEmpty := TRUE;
	                "Pallets_Stations".Stations[#i, #j].IsOccupied := FALSE;
	            ELSE
	                // Unknown state
	                "Pallets_Stations".Stations[#i, #j].IsEmpty := FALSE;
	                "Pallets_Stations".Stations[#i, #j].IsOccupied := FALSE;
	            END_IF;
	        END_FOR;
	    END_FOR;
	    
	END_REGION
	
END_FUNCTION_BLOCK

FUNCTION_BLOCK "SideShifter_Alarms"
{ S7_Optimized_Access := 'TRUE' }
VERSION : 0.1

BEGIN
END_FUNCTION_BLOCK

DATA_BLOCK "Main_Safety_RTG1_DB"   // DB6, F_DB
NAME : FUSI
// stored: InstanceOfName Main_Safety_RTG1, InstanceOfType FB
"Main_Safety_RTG1"
BEGIN
END_DATA_BLOCK

DATA_BLOCK "DB_SideShifter_1"   // DB2
// stored: InstanceOfName SideShifter, InstanceOfType FB
"SideShifter"
BEGIN
END_DATA_BLOCK

DATA_BLOCK "InstAnalyzeTokens"   // DB4
{ DB_Accessible_From_OPC_UA := 'FALSE' }
AUTHOR : SIEMENS AG
VERSION : 3.0
// stored: DBAccessibleFromOPCUA false, InstanceOfName AnalyzeTokens, InstanceOfType FB
"AnalyzeTokens"
   // VAR_INPUT
   //    tdsTelegramArrayLength { ExternalAccessible := 'False'; ExternalVisible := 'False'; ExternalWritable := 'False'} : UDInt;
   //    execute { ExternalAccessible := 'False'; ExternalVisible := 'False'; ExternalWritable := 'False'} : Bool;
   // END_VAR
   // VAR_OUTPUT
   //    status { ExternalAccessible := 'False'; ExternalVisible := 'False'; ExternalWritable := 'False'} : Word;
   //    error { ExternalAccessible := 'False'; ExternalVisible := 'False'; ExternalWritable := 'False'} : Bool;
   //    busy { ExternalAccessible := 'False'; ExternalVisible := 'False'; ExternalWritable := 'False'} : Bool;
   //    done { ExternalAccessible := 'False'; ExternalVisible := 'False'; ExternalWritable := 'False'} : Bool;
   //    metaDataAndRowsAvailable { ExternalAccessible := 'False'; ExternalVisible := 'False'; ExternalWritable := 'False'} : Bool;
   //    tdsHeader { ExternalAccessible := 'False'; ExternalVisible := 'False'; ExternalWritable := 'False'} : "LSql_typePacketHeader";
   //    columnCount { ExternalAccessible := 'False'; ExternalVisible := 'False'; ExternalWritable := 'False'} : UInt;
   //    rowCount { ExternalAccessible := 'False'; ExternalVisible := 'False'; ExternalWritable := 'False'} : UDInt;
   //    rowDataStart { ExternalAccessible := 'False'; ExternalVisible := 'False'; ExternalWritable := 'False'} : UInt;
   //    rowDataLength { ExternalAccessible := 'False'; ExternalVisible := 'False'; ExternalWritable := 'False'} : UDInt;
   //    errorToken { ExternalAccessible := 'False'; ExternalVisible := 'False'; ExternalWritable := 'False'} : "LSql_typeErrorToken";
   // END_VAR
   // VAR_IN_OUT
   //    tdsTelegramArray : Array[*] of Byte;
   //    columns : Array[*] of "LSql_typeColumn";
   // END_VAR
   // VAR
   //    statDone { ExternalAccessible := 'False'; ExternalVisible := 'False'; ExternalWritable := 'False'} : Bool;
   //    statError { ExternalAccessible := 'False'; ExternalVisible := 'False'; ExternalWritable := 'False'} : Bool;
   //    statBusy { ExternalAccessible := 'False'; ExternalVisible := 'False'; ExternalWritable := 'False'} : Bool;
   //    statRowsAvailable { ExternalAccessible := 'False'; ExternalVisible := 'False'; ExternalWritable := 'False'} : Bool;
   //    statMetaDataAvailable { ExternalAccessible := 'False'; ExternalVisible := 'False'; ExternalWritable := 'False'} : Bool;
   // END_VAR
BEGIN
END_DATA_BLOCK

DATA_BLOCK "InstDeserializeRows"   // DB9
{ DB_Accessible_From_OPC_UA := 'FALSE' }
// stored: DBAccessibleFromOPCUA false, InstanceOfName DeserializeRows, InstanceOfType FB
"DeserializeRows"
   // VAR_INPUT
   //    columnCount { ExternalAccessible := 'False'; ExternalVisible := 'False'; ExternalWritable := 'False'} : UInt;
   //    columns { ExternalAccessible := 'False'; ExternalVisible := 'False'; ExternalWritable := 'False'} : Array[0.."LSQL_NUMBER_OF_COLUMNS_MAX"] of "LSql_typeColumn";
   //    rowCount { ExternalAccessible := 'False'; ExternalVisible := 'False'; ExternalWritable := 'False'} : UDInt;
   //    rowDataStart { ExternalAccessible := 'False'; ExternalVisible := 'False'; ExternalWritable := 'False'} : UInt;
   //    rowDataLength { ExternalAccessible := 'False'; ExternalVisible := 'False'; ExternalWritable := 'False'} : UDInt;
   //    numberOfRowsPerCycle { ExternalAccessible := 'False'; ExternalVisible := 'False'; ExternalWritable := 'False'} : USInt;
   //    execute { ExternalAccessible := 'False'; ExternalVisible := 'False'; ExternalWritable := 'False'} : Bool;
   // END_VAR
   // VAR_OUTPUT
   //    busy { ExternalAccessible := 'False'; ExternalVisible := 'False'; ExternalWritable := 'False'} : Bool;
   //    done { ExternalAccessible := 'False'; ExternalVisible := 'False'; ExternalWritable := 'False'} : Bool;
   //    error { ExternalAccessible := 'False'; ExternalVisible := 'False'; ExternalWritable := 'False'} : Bool;
   //    warning { ExternalAccessible := 'False'; ExternalVisible := 'False'; ExternalWritable := 'False'} : Bool;
   //    rowOverflow { ExternalAccessible := 'False'; ExternalVisible := 'False'; ExternalWritable := 'False'} : Bool;
   //    status { ExternalAccessible := 'False'; ExternalVisible := 'False'; ExternalWritable := 'False'} : Word;
   // END_VAR
   // VAR_IN_OUT
   //    tdsTelegramArray : Array[*] of Byte;
   //    rows : Array[*] of "typeTokenRow";
   // END_VAR
   // VAR
   //    statRowOverflow { ExternalAccessible := 'False'; ExternalVisible := 'False'; ExternalWritable := 'False'} : Bool;
   //    statBusy { ExternalAccessible := 'False'; ExternalVisible := 'False'; ExternalWritable := 'False'} : Bool;
   //    statDone { ExternalAccessible := 'False'; ExternalVisible := 'False'; ExternalWritable := 'False'} : Bool;
   //    statError { ExternalAccessible := 'False'; ExternalVisible := 'False'; ExternalWritable := 'False'} : Bool;
   //    statWarning { ExternalAccessible := 'False'; ExternalVisible := 'False'; ExternalWritable := 'False'} : Bool;
   //    statStatus { ExternalAccessible := 'False'; ExternalVisible := 'False'; ExternalWritable := 'False'} : Word;
   //    statRowsDeserialized { ExternalAccessible := 'False'; ExternalVisible := 'False'; ExternalWritable := 'False'} : UDInt;
   //    statByteAddressCounter { ExternalAccessible := 'False'; ExternalVisible := 'False'; ExternalWritable := 'False'} : DInt;
   // END_VAR
BEGIN
END_DATA_BLOCK

DATA_BLOCK "InstLSql_Microsoft"   // DB1
{ DB_Accessible_From_OPC_UA := 'FALSE' }
AUTHOR : (department/personInCharge/contact)
FAMILY : (family)
// stored: AutoNumber false, DBAccessibleFromOPCUA false, InstanceOfName LSql_Microsoft, InstanceOfType FB
"LSql_Microsoft"
   // VAR_INPUT
   //    enable { ExternalAccessible := 'False'; ExternalVisible := 'False'; ExternalWritable := 'False'} : Bool;
   //    connectionSettings { ExternalAccessible := 'False'; ExternalVisible := 'False'; ExternalWritable := 'False'} : "LSql_typeConnectionSettings";
   //    command { ExternalAccessible := 'False'; ExternalVisible := 'False'; ExternalWritable := 'False'} : String;
   //    executeCommand { ExternalAccessible := 'False'; ExternalVisible := 'False'; ExternalWritable := 'False'} : Bool;
   // END_VAR
   // VAR_OUTPUT
   //    valid { ExternalWritable := 'False'} : Bool;
   //    busy { ExternalWritable := 'False'} : Bool;
   //    error { ExternalWritable := 'False'} : Bool;
   //    status { ExternalWritable := 'False'} : Word;
   //    diagnostics { ExternalWritable := 'False'} : "LSql_typeDiagnostics";
   //    dataReceived { ExternalWritable := 'False'} : Bool;
   //    tdsTelegramArrayLength { ExternalWritable := 'False'} : UDInt;
   // END_VAR
   // VAR_IN_OUT
   //    tdsTelegramArray : Array[*] of Byte;
   // END_VAR
   // VAR
   //    instTsend { ExternalAccessible := 'False'; ExternalVisible := 'False'; ExternalWritable := 'False'} : TSEND;
   //    instTcon { ExternalAccessible := 'False'; ExternalVisible := 'False'; ExternalWritable := 'False'} : TCON;
   //    instTrcv { ExternalAccessible := 'False'; ExternalVisible := 'False'; ExternalWritable := 'False'} : TRCV;
   //    instTdiscon { ExternalAccessible := 'False'; ExternalVisible := 'False'; ExternalWritable := 'False'} : TDISCON;
   //    statEnableOld { ExternalAccessible := 'False'; ExternalVisible := 'False'; ExternalWritable := 'False'} : Bool;
   //    statEnable { ExternalAccessible := 'False'; ExternalVisible := 'False'; ExternalWritable := 'False'} : Bool;
   //    statValid { ExternalAccessible := 'False'; ExternalVisible := 'False'; ExternalWritable := 'False'} : Bool;
   //    statBusy { ExternalAccessible := 'False'; ExternalVisible := 'False'; ExternalWritable := 'False'} : Bool;
   //    statError { ExternalAccessible := 'False'; ExternalVisible := 'False'; ExternalWritable := 'False'} : Bool;
   //    statErrorUserCleared { ExternalAccessible := 'False'; ExternalVisible := 'False'; ExternalWritable := 'False'} : Bool;
   //    statErrorAutoCleared { ExternalAccessible := 'False'; ExternalVisible := 'False'; ExternalWritable := 'False'} : Bool;
   //    statStatus { ExternalAccessible := 'False'; ExternalVisible := 'False'; ExternalWritable := 'False'} : Word;
   //    statSubfunctionStatus { ExternalAccessible := 'False'; ExternalVisible := 'False'; ExternalWritable := 'False'} : Word;
   //    statFBErrorState { ExternalAccessible := 'False'; ExternalVisible := 'False'; ExternalWritable := 'False'} : DInt;
   //    statFBState { ExternalAccessible := 'False'; ExternalVisible := 'False'; ExternalWritable := 'False'} : DInt;
   //    statDisablingCompleted { ExternalAccessible := 'False'; ExternalVisible := 'False'; ExternalWritable := 'False'} : Bool;
   //    statEmptyDiagnostics { ExternalAccessible := 'False'; ExternalVisible := 'False'; ExternalWritable := 'False'} : "LSql_typeDiagnostics";
   //    statReceivedBytes { ExternalAccessible := 'False'; ExternalVisible := 'False'; ExternalWritable := 'False'} : UDInt;
   //    statExecuteSqlBatchOld { ExternalAccessible := 'False'; ExternalVisible := 'False'; ExternalWritable := 'False'} : Bool;
   //    statSqlBatchData { ExternalAccessible := 'False'; ExternalVisible := 'False'; ExternalWritable := 'False'} : "LSql_typeSqlBatchData";
   //    statSqlBatch { ExternalAccessible := 'False'; ExternalVisible := 'False'; ExternalWritable := 'False'} : Array[0..2047] of Byte;
   //    statSqlBatchLen { ExternalAccessible := 'False'; ExternalVisible := 'False'; ExternalWritable := 'False'} : DInt;
   //    statWriter { ExternalAccessible := 'False'; ExternalVisible := 'False'; ExternalWritable := 'False'} : Int;
   //    statStatusSqlBatchIntToWord { ExternalAccessible := 'False'; ExternalVisible := 'False'; ExternalWritable := 'False'} : Word;
   //    statLoginData { ExternalAccessible := 'False'; ExternalVisible := 'False'; ExternalWritable := 'False'} : "LSql_typeLoginData";
   //    statLogin { ExternalAccessible := 'False'; ExternalVisible := 'False'; ExternalWritable := 'False'} : Array[0..2047] of Byte;
   //    statLoginLen { ExternalAccessible := 'False'; ExternalVisible := 'False'; ExternalWritable := 'False'} : DInt;
   //    statStatusLoginIntToWord { ExternalAccessible := 'False'; ExternalVisible := 'False'; ExternalWritable := 'False'} : Word;
   //    statStatusPreLoginIntToWord { ExternalAccessible := 'False'; ExternalVisible := 'False'; ExternalWritable := 'False'} : Word;
   //    statPreLogin { ExternalAccessible := 'False'; ExternalVisible := 'False'; ExternalWritable := 'False'} : Array[0..2047] of Byte;
   //    statPreLoginLen { ExternalAccessible := 'False'; ExternalVisible := 'False'; ExternalWritable := 'False'} : DInt;
   //    statPreLoginCache { ExternalAccessible := 'False'; ExternalVisible := 'False'; ExternalWritable := 'False'} : Array[0..2047] of Byte;
   //    statPreLoginData { ExternalAccessible := 'False'; ExternalVisible := 'False'; ExternalWritable := 'False'} : "LSql_typePreloginData";
   //    statErrorWriteData { ExternalAccessible := 'False'; ExternalVisible := 'False'; ExternalWritable := 'False'} : Bool;
   //    statWriteData { ExternalAccessible := 'False'; ExternalVisible := 'False'; ExternalWritable := 'False'} : Word;
   //    statTransmissionSqlCommand { ExternalAccessible := 'False'; ExternalVisible := 'False'; ExternalWritable := 'False'} : Bool;
   //    statTdsDataReceived { ExternalAccessible := 'False'; ExternalVisible := 'False'; ExternalWritable := 'False'} : Bool;
   //    statTdsTelegramBytesReceived { ExternalAccessible := 'False'; ExternalVisible := 'False'; ExternalWritable := 'False'} : UDInt;
   //    statTdsFragmBufferBytesFilled { ExternalAccessible := 'False'; ExternalVisible := 'False'; ExternalWritable := 'False'} : UDInt;
   //    statTdsFragmHeaderBytesFilled { ExternalAccessible := 'False'; ExternalVisible := 'False'; ExternalWritable := 'False'} : UDInt;
   //    statTdsFragmLengthFromHeader { ExternalAccessible := 'False'; ExternalVisible := 'False'; ExternalWritable := 'False'} : UDInt;
   //    statTdsTelegramLength { ExternalAccessible := 'False'; ExternalVisible := 'False'; ExternalWritable := 'False'} : UDInt;
   //    statTdsFragmStatus { ExternalAccessible := 'False'; ExternalVisible := 'False'; ExternalWritable := 'False'} : Byte;
   //    statTrcvBlockBufferArray { ExternalAccessible := 'False'; ExternalVisible := 'False'; ExternalWritable := 'False'} : Array[0..2047] of Byte;
   //    statTdsFragmHeaderBuffer { ExternalAccessible := 'False'; ExternalVisible := 'False'; ExternalWritable := 'False'} : Array[0..7] of Byte;
   //    statTdsTelegramContinuing { ExternalAccessible := 'False'; ExternalVisible := 'False'; ExternalWritable := 'False'} : Bool;
   //    statTdsTelegramArrayLowerBound { ExternalAccessible := 'False'; ExternalVisible := 'False'; ExternalWritable := 'False'} : DInt;
   //    statTdsTelegramArrayUpperBound { ExternalAccessible := 'False'; ExternalVisible := 'False'; ExternalWritable := 'False'} : DInt;
   // END_VAR
BEGIN
END_DATA_BLOCK

DATA_BLOCK "CS_Drive_PL"   // DB10, Motion_DB
// stored: InstanceOfName TO_SynchronousAxis, OfSystemLibElement TO_SynchronousAxis, OfSystemLibVersion 7.0
TO_SynchronousAxis   // technology object, version 7.0
// stored: Connection Interface Actor, InputAddress 400, OutputAddress 400
// stored: Connection Interface Sensor[1], InputAddress 400, OutputAddress 400, SensorIndexInActorTelegram 1
   // // inherited from TO_PositioningAxis
   // // inherited from TO_SpeedAxis
   // // inherited from TO_Axis
   // // inherited from TO_Object
   // VAR
   //    Actor : TO_Struct_Actor;
   // END_VAR
   // VAR
   //    Sensor : Array[1..4] of TO_Struct_Sensor;
   //    PositionControl : TO_Struct_PositionControl;
   // END_VAR
   // VAR
   //    StatusSynchronizedMotion { ExternalWritable := 'False'; S7_SetPoint := 'True'} : TO_Struct_StatusSynchronizedMotion;
   // END_VAR
BEGIN
   Actor.Interface.AddressIn.RID := 16#208072a;
   Actor.Interface.AddressIn.AREA := 16#81;
   Actor.Interface.AddressIn.OFFSET := 400;
   Actor.Interface.AddressOut.RID := 16#208072b;
   Actor.Interface.AddressOut.AREA := 16#82;
   Actor.Interface.AddressOut.OFFSET := 400;
   Sensor[1].Interface.AddressIn.RID := 16#208072a;
   Sensor[1].Interface.AddressIn.AREA := 16#81;
   Sensor[1].Interface.AddressIn.OFFSET := 400;
   Sensor[1].Interface.AddressOut.RID := 16#208072b;
   Sensor[1].Interface.AddressOut.AREA := 16#82;
   Sensor[1].Interface.AddressOut.OFFSET := 400;
   PositionControl.EnableDSC := true;
   _Actor.Interface.Telegram := 105;
   _Sensor[1].Interface.Telegram := 105;
END_DATA_BLOCK

DATA_BLOCK "CS_Drive_PP"   // DB12, Motion_DB
// stored: InstanceOfName TO_SynchronousAxis, OfSystemLibElement TO_SynchronousAxis, OfSystemLibVersion 7.0
TO_SynchronousAxis   // technology object, version 7.0
// stored: Connection Interface Actor, InputAddress 144, OutputAddress 144
// stored: Connection Interface Sensor[1], InputAddress 144, OutputAddress 144, SensorIndexInActorTelegram 1
   // // inherited from TO_PositioningAxis
   // // inherited from TO_SpeedAxis
   // // inherited from TO_Axis
   // // inherited from TO_Object
   // VAR
   //    Actor : TO_Struct_Actor;
   // END_VAR
   // VAR
   //    Sensor : Array[1..4] of TO_Struct_Sensor;
   //    PositionControl : TO_Struct_PositionControl;
   // END_VAR
   // VAR
   //    StatusSynchronizedMotion { ExternalWritable := 'False'; S7_SetPoint := 'True'} : TO_Struct_StatusSynchronizedMotion;
   // END_VAR
BEGIN
   Actor.Interface.AddressIn.RID := 16#208072a;
   Actor.Interface.AddressIn.AREA := 16#81;
   Actor.Interface.AddressIn.OFFSET := 144;
   Actor.Interface.AddressOut.RID := 16#208072b;
   Actor.Interface.AddressOut.AREA := 16#82;
   Actor.Interface.AddressOut.OFFSET := 144;
   Sensor[1].Interface.AddressIn.RID := 16#208072a;
   Sensor[1].Interface.AddressIn.AREA := 16#81;
   Sensor[1].Interface.AddressIn.OFFSET := 144;
   Sensor[1].Interface.AddressOut.RID := 16#208072b;
   Sensor[1].Interface.AddressOut.AREA := 16#82;
   Sensor[1].Interface.AddressOut.OFFSET := 144;
   PositionControl.EnableDSC := true;
   _Actor.Interface.Telegram := 105;
   _Sensor[1].Interface.Telegram := 105;
END_DATA_BLOCK

